C07146=1020.589,122.542,-113.459,167.523,51.122,159.470
C07147=1020.584,122.293,-113.440,167.519,51.128,159.471
C07148=1020.579,122.044,-113.421,167.517,51.134,159.471
C07149=1020.573,121.794,-113.402,167.514,51.141,159.472
C07150=1020.568,121.546,-113.383,167.511,51.148,159.473
C07151=1020.562,121.296,-113.363,167.508,51.155,159.474
C07152=1020.556,121.047,-113.344,167.505,51.160,159.475
C07153=1020.551,120.798,-113.325,167.502,51.167,159.475
C07154=1020.546,120.549,-113.306,167.500,51.174,159.476
C07155=1020.541,120.300,-113.287,167.497,51.180,159.477
C07156=1020.536,120.050,-113.267,167.494,51.187,159.478
C07157=1020.530,119.801,-113.248,167.491,51.193,159.478
C07158=1020.525,119.552,-113.229,167.488,51.200,159.479
C07159=1020.519,119.302,-113.210,167.485,51.207,159.480
C07160=1020.514,119.054,-113.191,167.482,51.214,159.481
C07161=1020.508,118.804,-113.172,167.479,51.219,159.482
C07162=1020.503,118.556,-113.153,167.476,51.226,159.482
C07163=1020.498,118.306,-113.134,167.474,51.233,159.483
C07164=1020.492,118.057,-113.114,167.470,51.240,159.484
C07165=1020.487,117.807,-113.096,167.468,51.246,159.485
C07166=1020.481,117.558,-113.077,167.464,51.253,159.485
C07167=1020.476,117.309,-113.058,167.462,51.259,159.486
C07168=1020.471,117.060,-113.039,167.459,51.266,159.487
C07169=1020.466,116.811,-113.019,167.456,51.272,159.488
C07170=1020.461,116.561,-113.000,167.453,51.278,159.489
C07171=1020.456,116.313,-112.981,167.450,51.285,159.489
C07172=1020.450,116.062,-112.963,167.447,51.291,159.490
C07173=1020.445,115.814,-112.944,167.444,51.298,159.491
C07174=1020.439,115.564,-112.925,167.442,51.305,159.492
C07175=1020.434,115.316,-112.906,167.439,51.311,159.492
C07176=1020.429,115.066,-112.887,167.436,51.317,159.493
C07177=1020.424,114.817,-112.868,167.433,51.324,159.494
C07178=1020.418,114.567,-112.849,167.430,51.331,159.495
C07179=1020.413,114.319,-112.830,167.427,51.337,159.495
C07180=1020.407,114.069,-112.811,167.424,51.344,159.496
C07181=1020.402,113.820,-112.792,167.422,51.350,159.497
C07182=1020.397,113.571,-112.773,167.419,51.356,159.498
C07183=1020.392,113.322,-112.755,167.416,51.363,159.498
C07184=1020.387,113.072,-112.735,167.413,51.370,159.499
C07185=1020.382,112.823,-112.716,167.411,51.376,159.500
C07186=1020.376,112.574,-112.697,167.407,51.383,159.501
C07187=1020.371,112.324,-112.679,167.405,51.389,159.502
C07188=1020.366,112.075,-112.659,167.401,51.395,159.502
C07189=1020.360,111.826,-112.642,167.399,51.402,159.503
C07190=1020.354,111.577,-112.623,167.395,51.409,159.504
C07191=1020.349,111.328,-112.604,167.393,51.415,159.505
C07192=1020.344,111.078,-112.585,167.390,51.422,159.505
C07193=1020.338,110.829,-112.567,167.387,51.428,159.506
C07194=1020.333,110.579,-112.548,167.385,51.435,159.507
C07195=1020.328,110.331,-112.530,167.382,51.442,159.508
C07196=1020.322,110.080,-112.511,167.379,51.448,159.509
C07197=1020.316,109.832,-112.493,167.376,51.455,159.509
C07198=1020.311,109.583,-112.474,167.373,51.461,159.510
C07199=1020.306,109.333,-112.455,167.370,51.468,159.511
C07200=1020.301,109.085,-112.436,167.368,51.475,159.512
C07201=1020.295,108.835,-112.418,167.364,51.482,159.512
C07202=1020.290,108.585,-112.400,167.362,51.488,159.513
C07203=1020.284,108.336,-112.382,167.359,51.495,159.514
C07204=1020.279,108.087,-112.364,167.356,51.502,159.515
C07205=1020.273,107.838,-112.344,167.353,51.508,159.516
C07206=1020.267,107.555,-112.324,167.350,51.516,159.517
C07207=1020.261,107.272,-112.303,167.347,51.523,159.518
C07208=1020.254,106.989,-112.282,167.344,51.531,159.518
C07209=1020.249,106.707,-112.262,167.341,51.539,159.519
C07210=1020.243,106.457,-112.243,167.337,51.545,159.520
C07211=1020.237,106.208,-112.225,167.335,51.551,159.521
C07212=1020.232,105.958,-112.206,167.332,51.558,159.522
C07213=1020.226,105.710,-112.188,167.329,51.565,159.523
C07214=1020.221,105.460,-112.170,167.326,51.572,159.523
C07215=1020.216,105.210,-112.151,167.324,51.579,159.524
C07216=1020.210,104.962,-112.133,167.321,51.584,159.525
C07217=1020.205,104.712,-112.115,167.318,51.591,159.526
C07218=1020.199,104.463,-112.097,167.316,51.598,159.526
C07219=1020.194,104.214,-112.078,167.312,51.605,159.527
C07220=1020.189,103.964,-112.060,167.310,51.611,159.528
C07221=1020.183,103.715,-112.042,167.306,51.618,159.529
C07222=1020.178,103.466,-112.023,167.304,51.624,159.530
C07223=1020.172,103.216,-112.005,167.302,51.631,159.530
C07224=1020.167,102.967,-111.987,167.298,51.638,159.531
C07225=1020.161,102.719,-111.969,167.296,51.644,159.532
C07226=1020.156,102.469,-111.950,167.292,51.651,159.533
C07227=1020.151,102.219,-111.932,167.290,51.658,159.533
C07228=1020.146,101.970,-111.915,167.288,51.664,159.534
C07229=1020.140,101.721,-111.895,167.284,51.670,159.535
C07230=1020.135,101.472,-111.878,167.282,51.677,159.536
C07231=1020.130,101.222,-111.860,167.279,51.684,159.537
C07232=1020.124,100.973,-111.842,167.276,51.691,159.537
C07233=1020.119,100.724,-111.823,167.274,51.697,159.538
C07234=1020.114,100.475,-111.805,167.270,51.704,159.539
C07235=1020.108,100.225,-111.787,167.268,51.710,159.540
C07236=1020.103,99.975,-111.768,167.266,51.717,159.541
C07237=1020.097,99.727,-111.750,167.262,51.723,159.541
C07238=1020.092,99.477,-111.732,167.260,51.730,159.542
C07239=1020.086,99.228,-111.714,167.257,51.737,159.543
C07240=1020.081,98.979,-111.696,167.254,51.743,159.544
C07241=1020.076,98.730,-111.678,167.252,51.749,159.544
C07242=1020.070,98.480,-111.660,167.248,51.756,159.545
C07243=1020.065,98.230,-111.642,167.246,51.763,159.546
C07244=1020.059,97.981,-111.625,167.243,51.770,159.547
C07245=1020.053,97.732,-111.607,167.241,51.776,159.548
C07246=1020.048,97.483,-111.589,167.237,51.783,159.548
C07247=1020.043,97.234,-111.570,167.235,51.790,159.549
C07248=1020.037,96.985,-111.553,167.231,51.796,159.550
C07249=1020.031,96.735,-111.535,167.229,51.803,159.551
C07250=1020.026,96.486,-111.517,167.227,51.810,159.552
C07251=1020.021,96.237,-111.499,167.224,51.817,159.552
C07252=1020.015,95.987,-111.481,167.221,51.823,159.553
C07253=1020.009,95.738,-111.464,167.218,51.830,159.554
C07254=1020.004,95.489,-111.445,167.215,51.836,159.555
C07255=1019.999,95.240,-111.428,167.213,51.843,159.556
C07256=1019.993,94.990,-111.410,167.210,51.850,159.556
C07257=1019.988,94.740,-111.392,167.208,51.857,159.557
C07258=1019.982,94.491,-111.374,167.204,51.863,159.558
C07259=1019.977,94.242,-111.357,167.202,51.869,159.559
C07260=1019.972,93.993,-111.340,167.200,51.876,159.559
C07261=1019.966,93.743,-111.321,167.196,51.883,159.560
C07262=1019.961,93.494,-111.304,167.194,51.890,159.561
C07263=1019.955,93.245,-111.286,167.190,51.896,159.562
C07264=1019.950,92.995,-111.268,167.188,51.903,159.563
C07265=1019.945,92.746,-111.250,167.186,51.909,159.563
C07266=1019.939,92.496,-111.232,167.183,51.916,159.564
C07267=1019.933,92.247,-111.215,167.180,51.922,159.565
C07268=1019.929,91.998,-111.197,167.177,51.929,159.566
C07269=1019.923,91.749,-111.179,167.175,51.936,159.567
C07270=1019.917,91.466,-111.159,167.171,51.943,159.567
C07271=1019.910,91.184,-111.139,167.169,51.951,159.568
C07272=1019.905,90.900,-111.119,167.166,51.958,159.569
C07273=1019.899,90.618,-111.099,167.162,51.965,159.570
C07274=1019.893,90.368,-111.081,167.159,51.972,159.571
C07275=1019.887,90.119,-111.064,167.157,51.979,159.572
C07276=1019.882,89.870,-111.045,167.154,51.985,159.572
C07277=1019.877,89.621,-111.028,167.151,51.992,159.573
C07278=1019.872,89.371,-111.011,167.149,51.999,159.574
C07279=1019.866,89.122,-110.993,167.146,52.005,159.575
C07280=1019.860,88.872,-110.975,167.143,52.012,159.575
C07281=1019.855,88.623,-110.958,167.141,52.018,159.576
C07282=1019.849,88.374,-110.941,167.139,52.025,159.577
C07283=1019.844,88.125,-110.923,167.135,52.032,159.578
C07284=1019.838,87.875,-110.906,167.133,52.039,159.579
C07285=1019.833,87.626,-110.889,167.130,52.046,159.580
C07286=1019.828,87.377,-110.871,167.127,52.052,159.580
C07287=1019.821,87.127,-110.854,167.124,52.059,159.581
C07288=1019.816,86.877,-110.837,167.122,52.065,159.582
C07289=1019.811,86.628,-110.819,167.120,52.072,159.583
C07290=1019.805,86.379,-110.802,167.116,52.079,159.583
C07291=1019.800,86.130,-110.785,167.114,52.085,159.584
C07292=1019.794,85.881,-110.767,167.111,52.092,159.585
C07293=1019.789,85.632,-110.750,167.108,52.099,159.586
C07294=1019.784,85.382,-110.733,167.106,52.106,159.587
C07295=1019.778,85.132,-110.715,167.103,52.113,159.587
C07296=1019.772,84.882,-110.698,167.100,52.119,159.588
C07297=1019.767,84.633,-110.680,167.097,52.126,159.589
C07298=1019.761,84.384,-110.663,167.095,52.132,159.590
C07299=1019.756,84.135,-110.646,167.093,52.139,159.591
C07300=1019.751,83.886,-110.628,167.089,52.145,159.591
C07301=1019.745,83.636,-110.612,167.087,52.152,159.592
C07302=1019.739,83.387,-110.595,167.085,52.159,159.593
C07303=1019.734,83.138,-110.578,167.081,52.166,159.594
C07304=1019.728,82.889,-110.560,167.079,52.172,159.594
C07305=1019.723,82.640,-110.543,167.076,52.179,159.595
C07306=1019.718,82.390,-110.526,167.073,52.185,159.596
C07307=1019.712,82.141,-110.508,167.071,52.192,159.597
C07308=1019.706,81.891,-110.491,167.068,52.198,159.597
C07309=1019.701,81.641,-110.473,167.065,52.205,159.598
C07310=1019.696,81.392,-110.457,167.063,52.212,159.599
C07311=1019.690,81.143,-110.439,167.060,52.218,159.600
C07312=1019.685,80.893,-110.422,167.057,52.225,159.601
C07313=1019.679,80.644,-110.405,167.055,52.232,159.602
C07314=1019.674,80.394,-110.388,167.052,52.239,159.602
C07315=1019.669,80.145,-110.370,167.049,52.245,159.603
C07316=1019.663,79.896,-110.353,167.047,52.251,159.604
C07317=1019.658,79.647,-110.336,167.044,52.258,159.605
C07318=1019.653,79.397,-110.319,167.041,52.264,159.605
C07319=1019.647,79.148,-110.301,167.039,52.271,159.606
C07320=1019.641,78.899,-110.285,167.036,52.278,159.607
C07321=1019.636,78.650,-110.267,167.033,52.284,159.608
C07322=1019.630,78.400,-110.251,167.031,52.291,159.608
C07323=1019.625,78.151,-110.233,167.028,52.297,159.609
C07324=1019.620,77.901,-110.216,167.026,52.304,159.610
C07325=1019.615,77.652,-110.199,167.023,52.311,159.611
C07326=1019.609,77.403,-110.182,167.021,52.317,159.611
C07327=1019.604,77.153,-110.165,167.018,52.324,159.612
C07328=1019.598,76.904,-110.147,167.015,52.330,159.613
C07329=1019.592,76.654,-110.131,167.013,52.336,159.614
C07330=1019.587,76.405,-110.114,167.010,52.343,159.615
C07331=1019.582,76.156,-110.097,167.007,52.350,159.615
C07332=1019.576,75.906,-110.080,167.004,52.357,159.616
C07333=1019.570,75.657,-110.064,167.002,52.363,159.617
C07334=1019.564,75.374,-110.045,166.999,52.371,159.618
C07335=1019.558,75.091,-110.026,166.996,52.379,159.619
C07336=1019.552,74.810,-110.006,166.993,52.386,159.620
C07337=1019.546,74.527,-109.987,166.990,52.394,159.621
C07338=1019.541,74.277,-109.970,166.987,52.401,159.621
C07339=1019.535,74.027,-109.954,166.984,52.407,159.622
C07340=1019.530,73.778,-109.937,166.982,52.413,159.623
C07341=1019.524,73.529,-109.920,166.979,52.421,159.624
C07342=1019.519,73.279,-109.903,166.977,52.427,159.624
C07343=1019.513,73.030,-109.887,166.974,52.433,159.625
C07344=1019.508,72.780,-109.870,166.971,52.440,159.626
C07345=1019.502,72.531,-109.853,166.969,52.447,159.627
C07346=1019.496,72.282,-109.836,166.965,52.453,159.627
C07347=1019.491,72.032,-109.819,166.963,52.460,159.628
C07348=1019.486,71.783,-109.802,166.961,52.467,159.629
C07349=1019.480,71.533,-109.786,166.958,52.473,159.630
C07350=1019.475,71.284,-109.770,166.955,52.480,159.631
C07351=1019.469,71.035,-109.753,166.953,52.487,159.631
C07352=1019.464,70.786,-109.736,166.950,52.493,159.632
C07353=1019.458,70.536,-109.719,166.948,52.500,159.633
C07354=1019.453,70.287,-109.703,166.945,52.507,159.634
C07355=1019.447,70.037,-109.686,166.942,52.513,159.634
C07356=1019.442,69.788,-109.669,166.940,52.520,159.635
C07357=1019.436,69.538,-109.653,166.938,52.526,159.636
C07358=1019.431,69.289,-109.636,166.934,52.533,159.637
C07359=1019.426,69.040,-109.620,166.932,52.540,159.637
C07360=1019.420,68.790,-109.603,166.930,52.546,159.638
C07361=1019.415,68.541,-109.586,166.926,52.553,159.639
C07362=1019.409,68.292,-109.569,166.924,52.559,159.640
C07363=1019.404,68.042,-109.552,166.922,52.566,159.641
C07364=1019.398,67.793,-109.536,166.918,52.573,159.641
C07365=1019.393,67.543,-109.519,166.916,52.579,159.642
C07366=1019.387,67.295,-109.503,166.914,52.586,159.643
C07367=1019.382,67.045,-109.487,166.910,52.592,159.644
C07368=1019.376,66.796,-109.470,166.908,52.599,159.644
C07369=1019.370,66.546,-109.455,166.906,52.606,159.645
C07370=1019.365,66.296,-109.438,166.903,52.612,159.646
C07371=1019.359,66.047,-109.422,166.900,52.619,159.647
C07372=1019.355,65.798,-109.405,166.898,52.626,159.648
C07373=1019.349,65.548,-109.389,166.895,52.632,159.648
C07374=1019.343,65.299,-109.372,166.893,52.639,159.649
C07375=1019.337,65.049,-109.356,166.891,52.646,159.650
C07376=1019.332,64.800,-109.339,166.887,52.653,159.651
C07377=1019.326,64.550,-109.323,166.885,52.659,159.651
C07378=1019.321,64.302,-109.307,166.882,52.666,159.652
C07379=1019.316,64.052,-109.290,166.880,52.673,159.653
C07380=1019.310,63.803,-109.274,166.877,52.679,159.654
C07381=1019.305,63.552,-109.258,166.874,52.686,159.654
C07382=1019.299,63.303,-109.241,166.871,52.692,159.655
C07383=1019.294,63.054,-109.225,166.869,52.699,159.656
C07384=1019.288,62.805,-109.209,166.866,52.706,159.657
C07385=1019.282,62.555,-109.192,166.864,52.713,159.658
C07386=1019.277,62.305,-109.177,166.860,52.719,159.658
C07387=1019.271,62.056,-109.161,166.858,52.726,159.659
C07388=1019.265,61.807,-109.145,166.856,52.733,159.660
C07389=1019.260,61.557,-109.129,166.853,52.740,159.661
C07390=1019.254,61.308,-109.113,166.851,52.746,159.662
C07391=1019.248,61.059,-109.097,166.848,52.754,159.662
C07392=1019.243,60.808,-109.080,166.845,52.760,159.663
C07393=1019.238,60.560,-109.065,166.842,52.767,159.664
C07394=1019.232,60.310,-109.048,166.840,52.774,159.665
C07395=1019.226,60.060,-109.033,166.838,52.780,159.666
C07396=1019.220,59.811,-109.016,166.835,52.787,159.666
C07397=1019.215,59.562,-109.001,166.832,52.793,159.667
C07398=1019.208,59.279,-108.983,166.830,52.801,159.668
C07399=1019.202,58.996,-108.964,166.826,52.810,159.669
C07400=1019.195,58.713,-108.946,166.823,52.817,159.670
C07401=1019.189,58.431,-108.928,166.820,52.825,159.671
C07402=1019.184,58.181,-108.912,166.818,52.831,159.672
C07403=1019.178,57.932,-108.896,166.815,52.838,159.672
C07404=1019.172,57.682,-108.880,166.812,52.845,159.673
C07405=1019.167,57.433,-108.864,166.809,52.852,159.674
C07406=1019.161,57.184,-108.848,166.807,52.858,159.675
C07407=1019.155,56.934,-108.833,166.805,52.865,159.675
C07408=1019.150,56.685,-108.817,166.802,52.872,159.676
C07409=1019.144,56.435,-108.801,166.800,52.878,159.677
C07410=1019.139,56.186,-108.785,166.796,52.885,159.677
C07411=1019.133,55.937,-108.770,166.794,52.892,159.678
C07412=1019.128,55.687,-108.754,166.792,52.898,159.679
C07413=1019.122,55.438,-108.737,166.788,52.905,159.680
C07414=1019.117,55.188,-108.722,166.786,52.912,159.681
C07415=1019.111,54.939,-108.705,166.784,52.918,159.682
C07416=1019.106,54.689,-108.690,166.781,52.925,159.682
C07417=1019.100,54.440,-108.674,166.779,52.932,159.683
C07418=1019.095,54.190,-108.658,166.775,52.939,159.684
C07419=1019.089,53.941,-108.642,166.773,52.945,159.684
C07420=1019.084,53.692,-108.627,166.771,52.952,159.685
C07421=1019.078,53.442,-108.611,166.768,52.959,159.686
C07422=1019.072,53.193,-108.595,166.765,52.965,159.687
C07423=1019.067,52.944,-108.579,166.763,52.972,159.688
C07424=1019.061,52.694,-108.564,166.760,52.979,159.688
C07425=1019.056,52.444,-108.547,166.758,52.985,159.689
C07426=1019.051,52.195,-108.532,166.755,52.992,159.690
C07427=1019.045,51.946,-108.515,166.752,52.998,159.690
C07428=1019.039,51.696,-108.500,166.750,53.005,159.691
C07429=1019.034,51.447,-108.484,166.747,53.012,159.692
C07430=1019.028,51.197,-108.468,166.744,53.018,159.693
C07431=1019.023,50.948,-108.453,166.742,53.025,159.694
C07432=1019.017,50.698,-108.437,166.739,53.032,159.694
C07433=1019.012,50.448,-108.421,166.737,53.038,159.695
C07434=1019.006,50.200,-108.406,166.735,53.045,159.696
C07435=1019.001,49.950,-108.390,166.731,53.052,159.697
C07436=1018.995,49.701,-108.374,166.729,53.058,159.697
C07437=1018.990,49.451,-108.359,166.727,53.064,159.698
C07438=1018.985,49.201,-108.342,166.724,53.072,159.699
C07439=1018.979,48.952,-108.327,166.721,53.078,159.700
C07440=1018.974,48.702,-108.311,166.719,53.085,159.700
C07441=1018.968,48.454,-108.295,166.715,53.091,159.701
C07442=1018.963,48.204,-108.280,166.713,53.098,159.702
C07443=1018.958,47.954,-108.264,166.711,53.104,159.703
C07444=1018.952,47.705,-108.248,166.708,53.111,159.703
C07445=1018.947,47.456,-108.233,166.705,53.117,159.704
C07446=1018.941,47.206,-108.217,166.703,53.124,159.705
C07447=1018.935,46.957,-108.201,166.701,53.130,159.706
C07448=1018.930,46.707,-108.186,166.698,53.137,159.706
C07449=1018.924,46.457,-108.170,166.695,53.143,159.707
C07450=1018.919,46.209,-108.155,166.693,53.150,159.708
C07451=1018.913,45.959,-108.139,166.690,53.157,159.708
C07452=1018.908,45.709,-108.124,166.688,53.164,159.709
C07453=1018.903,45.460,-108.107,166.685,53.170,159.710
C07454=1018.898,45.210,-108.092,166.682,53.177,159.711
C07455=1018.892,44.961,-108.076,166.680,53.183,159.711
C07456=1018.887,44.712,-108.060,166.678,53.190,159.712
C07457=1018.881,44.462,-108.045,166.675,53.196,159.713
C07458=1018.876,44.213,-108.030,166.672,53.202,159.713
C07459=1018.870,43.963,-108.013,166.670,53.209,159.714
C07460=1018.865,43.714,-107.998,166.667,53.215,159.715
C07461=1018.860,43.464,-107.983,166.664,53.222,159.716
C07462=1018.854,43.182,-107.965,166.661,53.230,159.717
C07463=1018.848,42.898,-107.947,166.658,53.237,159.717
C07464=1018.842,42.616,-107.930,166.655,53.244,159.718
C07465=1018.835,42.333,-107.912,166.653,53.252,159.719
C07466=1018.830,42.083,-107.897,166.650,53.258,159.720
C07467=1018.824,41.833,-107.881,166.648,53.265,159.721
C07468=1018.819,41.584,-107.866,166.644,53.271,159.721
C07469=1018.814,41.335,-107.852,166.642,53.278,159.722
C07470=1018.808,41.085,-107.836,166.640,53.284,159.723
C07471=1018.803,40.836,-107.820,166.637,53.292,159.723
C07472=1018.797,40.586,-107.805,166.635,53.298,159.724
C07473=1018.792,40.337,-107.790,166.632,53.305,159.725
C07474=1018.786,40.088,-107.775,166.629,53.312,159.726
C07475=1018.781,39.838,-107.759,166.627,53.318,159.726
C07476=1018.775,39.588,-107.744,166.624,53.325,159.727
C07477=1018.770,39.339,-107.729,166.621,53.331,159.728
C07478=1018.763,39.089,-107.714,166.619,53.338,159.729
C07479=1018.758,38.840,-107.699,166.616,53.345,159.729
C07480=1018.753,38.591,-107.683,166.614,53.351,159.730
C07481=1018.748,38.341,-107.668,166.611,53.358,159.731
C07482=1018.742,38.092,-107.653,166.608,53.365,159.732
C07483=1018.736,37.842,-107.638,166.606,53.371,159.732
C07484=1018.731,37.593,-107.623,166.604,53.378,159.733
C07485=1018.726,37.343,-107.607,166.600,53.384,159.734
C07486=1018.721,37.093,-107.592,166.598,53.391,159.735
C07487=1018.715,36.845,-107.577,166.596,53.397,159.735
C07488=1018.709,36.595,-107.562,166.593,53.404,159.736
C07489=1018.704,36.345,-107.547,166.591,53.411,159.737
C07490=1018.698,36.096,-107.532,166.587,53.418,159.738
C07491=1018.693,35.846,-107.517,166.585,53.424,159.738
C07492=1018.687,35.597,-107.503,166.583,53.431,159.739
C07493=1018.682,35.347,-107.487,166.580,53.437,159.740
C07494=1018.676,35.098,-107.472,166.578,53.444,159.741
C07495=1018.671,34.849,-107.457,166.575,53.451,159.741
C07496=1018.664,34.599,-107.442,166.572,53.458,159.742
C07497=1018.660,34.349,-107.428,166.569,53.465,159.743
C07498=1018.653,34.099,-107.413,166.567,53.471,159.743
C07499=1018.648,33.850,-107.398,166.565,53.478,159.744
C07500=1018.642,33.601,-107.383,166.561,53.484,159.745
C07501=1018.637,33.351,-107.368,166.559,53.491,159.746
C07502=1018.631,33.102,-107.354,166.556,53.498,159.746
C07503=1018.626,32.852,-107.339,166.554,53.504,159.747
C07504=1018.620,32.603,-107.324,166.552,53.511,159.748
C07505=1018.615,32.353,-107.309,166.548,53.518,159.749
C07506=1018.609,32.104,-107.295,166.546,53.525,159.749
C07507=1018.604,31.854,-107.279,166.543,53.531,159.750
C07508=1018.598,31.605,-107.265,166.541,53.538,159.751
C07509=1018.593,31.356,-107.249,166.538,53.544,159.752
C07510=1018.588,31.105,-107.235,166.535,53.552,159.752
C07511=1018.582,30.856,-107.220,166.533,53.558,159.753
C07512=1018.577,30.607,-107.205,166.530,53.565,159.754
C07513=1018.570,30.357,-107.190,166.528,53.571,159.754
C07514=1018.566,30.107,-107.175,166.525,53.577,159.755
C07515=1018.560,29.858,-107.161,166.522,53.584,159.756
C07516=1018.555,29.609,-107.146,166.520,53.591,159.757
C07517=1018.549,29.359,-107.131,166.518,53.598,159.757
C07518=1018.544,29.110,-107.116,166.514,53.604,159.758
C07519=1018.538,28.861,-107.102,166.512,53.611,159.759
C07520=1018.532,28.610,-107.087,166.509,53.617,159.759
C07521=1018.527,28.361,-107.072,166.507,53.624,159.760
C07522=1018.522,28.112,-107.057,166.505,53.630,159.761
C07523=1018.516,27.862,-107.043,166.501,53.637,159.761
C07524=1018.511,27.612,-107.028,166.499,53.644,159.762
C07525=1018.505,27.363,-107.013,166.497,53.650,159.763
C07526=1018.499,27.089,-106.997,166.494,53.658,159.764
C07527=1018.492,26.814,-106.981,166.491,53.665,159.765
C07528=1018.486,26.539,-106.965,166.488,53.673,159.766
C07529=1018.480,26.265,-106.949,166.485,53.680,159.766
C07530=1018.475,26.007,-106.935,166.482,53.687,159.767
C07531=1018.469,25.749,-106.919,166.479,53.694,159.768
C07532=1018.463,25.491,-106.904,166.477,53.701,159.769
C07533=1018.457,25.233,-106.890,166.474,53.708,159.769
C07534=1018.452,24.984,-106.875,166.471,53.714,159.770
C07535=1018.447,24.734,-106.861,166.468,53.721,159.771
C07536=1018.441,24.485,-106.846,166.466,53.727,159.771
C07537=1018.435,24.235,-106.832,166.463,53.735,159.772
C07538=1018.430,23.985,-106.817,166.461,53.741,159.773
C07539=1018.424,23.736,-106.803,166.459,53.748,159.774
C07540=1018.419,23.487,-106.788,166.455,53.754,159.774
C07541=1018.413,23.237,-106.774,166.453,53.761,159.775
C07542=1018.408,22.987,-106.760,166.450,53.768,159.776
C07543=1018.402,22.738,-106.745,166.448,53.775,159.777
C07544=1018.397,22.488,-106.731,166.444,53.781,159.777
C07545=1018.391,22.239,-106.717,166.443,53.788,159.778
C07546=1018.386,21.989,-106.702,166.440,53.794,159.779
C07547=1018.380,21.739,-106.688,166.437,53.802,159.779
C07548=1018.374,21.490,-106.673,166.435,53.808,159.780
C07549=1018.369,21.241,-106.659,166.431,53.814,159.781
C07550=1018.364,20.991,-106.644,166.429,53.821,159.782
C07551=1018.358,20.742,-106.630,166.427,53.827,159.782
C07552=1018.353,20.492,-106.616,166.424,53.835,159.783
C07553=1018.347,20.243,-106.602,166.422,53.841,159.784
C07554=1018.342,19.993,-106.587,166.419,53.848,159.784
C07555=1018.336,19.743,-106.573,166.416,53.854,159.785
C07556=1018.330,19.494,-106.559,166.414,53.860,159.786
C07557=1018.325,19.245,-106.545,166.411,53.868,159.786
C07558=1018.320,18.995,-106.530,166.409,53.874,159.787
C07559=1018.314,18.746,-106.516,166.406,53.881,159.788
C07560=1018.309,18.496,-106.502,166.403,53.887,159.789
C07561=1018.303,18.246,-106.488,166.400,53.894,159.789
C07562=1018.297,17.996,-106.474,166.398,53.901,159.790
C07563=1018.292,17.747,-106.459,166.394,53.908,159.791
C07564=1018.286,17.498,-106.445,166.393,53.914,159.791
C07565=1018.281,17.248,-106.431,166.390,53.921,159.792
C07566=1018.275,16.999,-106.418,166.387,53.928,159.793
C07567=1018.269,16.750,-106.403,166.385,53.934,159.794
C07568=1018.265,16.500,-106.389,166.382,53.941,159.794
C07569=1018.259,16.250,-106.375,166.380,53.948,159.795
C07570=1018.254,16.001,-106.361,166.376,53.954,159.795
C07571=1018.248,15.751,-106.347,166.374,53.961,159.796
C07572=1018.242,15.501,-106.333,166.371,53.968,159.797
C07573=1018.236,15.252,-106.318,166.369,53.975,159.798
C07574=1018.231,15.002,-106.304,166.367,53.981,159.798
C07575=1018.225,14.753,-106.290,166.363,53.987,159.799
C07576=1018.220,14.503,-106.277,166.361,53.994,159.800
C07577=1018.214,14.253,-106.263,166.358,54.001,159.800
C07578=1018.209,14.004,-106.249,166.355,54.007,159.801
C07579=1018.204,13.755,-106.234,166.352,54.014,159.802
C07580=1018.198,13.505,-106.220,166.350,54.021,159.803
C07581=1018.193,13.255,-106.206,166.348,54.027,159.803
C07582=1018.187,13.006,-106.192,166.345,54.034,159.804
C07583=1018.181,12.757,-106.179,166.343,54.041,159.805
C07584=1018.176,12.507,-106.165,166.339,54.048,159.805
C07585=1018.170,12.258,-106.151,166.337,54.055,159.806
C07586=1018.165,12.008,-106.137,166.334,54.061,159.807
C07587=1018.159,11.758,-106.123,166.331,54.069,159.808
C07588=1018.153,11.509,-106.110,166.329,54.075,159.808
C07589=1018.148,11.259,-106.097,166.326,54.082,159.809
C07590=1018.142,10.977,-106.081,166.323,54.089,159.810
C07591=1018.135,10.696,-106.066,166.320,54.097,159.811
C07592=1018.129,10.415,-106.050,166.318,54.105,159.812
C07593=1018.123,10.133,-106.035,166.314,54.112,159.812
C07594=1018.117,9.884,-106.021,166.311,54.119,159.813
C07595=1018.111,9.634,-106.007,166.308,54.126,159.814
C07596=1018.106,9.385,-105.994,166.306,54.132,159.814
C07597=1018.100,9.135,-105.980,166.303,54.140,159.815
C07598=1018.095,8.886,-105.966,166.301,54.146,159.816
C07599=1018.090,8.636,-105.953,166.298,54.153,159.816
C07600=1018.083,8.386,-105.939,166.296,54.159,159.817
C07601=1018.078,8.137,-105.926,166.293,54.167,159.818
C07602=1018.073,7.887,-105.912,166.290,54.173,159.819
C07603=1018.067,7.638,-105.898,166.287,54.179,159.819
C07604=1018.061,7.388,-105.885,166.285,54.186,159.820
C07605=1018.056,7.138,-105.871,166.282,54.193,159.820
C07606=1018.050,6.888,-105.858,166.280,54.200,159.821
C07607=1018.045,6.639,-105.844,166.276,54.207,159.822
C07608=1018.039,6.389,-105.830,166.274,54.213,159.823
C07609=1018.034,6.141,-105.817,166.271,54.220,159.823
C07610=1018.028,5.891,-105.803,166.269,54.226,159.824
C07611=1018.023,5.641,-105.790,166.265,54.233,159.825
C07612=1018.017,5.391,-105.776,166.264,54.240,159.825
C07613=1018.012,5.142,-105.762,166.260,54.247,159.826
C07614=1018.006,4.893,-105.749,166.258,54.253,159.827
C07615=1018.000,4.643,-105.735,166.255,54.260,159.827
C07616=1017.995,4.393,-105.722,166.253,54.266,159.828
C07617=1017.990,4.143,-105.708,166.250,54.273,159.829
C07618=1017.984,3.894,-105.694,166.247,54.280,159.829
C07619=1017.979,3.645,-105.681,166.245,54.286,159.830
C07620=1017.973,3.395,-105.668,166.242,54.293,159.831
C07621=1017.968,3.145,-105.654,166.240,54.300,159.832
C07622=1017.962,2.896,-105.640,166.236,54.306,159.832
C07623=1017.957,2.646,-105.628,166.234,54.313,159.833
C07624=1017.951,2.396,-105.614,166.231,54.320,159.834
C07625=1017.946,2.147,-105.600,166.229,54.326,159.834
C07626=1017.941,1.898,-105.587,166.225,54.333,159.835
C07627=1017.936,1.648,-105.573,166.223,54.339,159.835
C07628=1017.929,1.398,-105.560,166.220,54.346,159.836
C07629=1017.924,1.149,-105.546,166.218,54.353,159.837
C07630=1017.919,0.899,-105.533,166.215,54.359,159.837
C07631=1017.913,0.649,-105.519,166.212,54.366,159.838
C07632=1017.908,0.401,-105.506,166.210,54.373,159.839
C07633=1017.902,0.150,-105.493,166.207,54.379,159.839
C07634=1017.897,-0.099,-105.479,166.205,54.385,159.840
C07635=1017.891,-0.349,-105.466,166.201,54.392,159.841
C07636=1017.886,-0.599,-105.452,166.199,54.398,159.841
C07637=1017.881,-0.848,-105.439,166.196,54.406,159.842
C07638=1017.875,-1.097,-105.426,166.194,54.412,159.843
C07639=1017.870,-1.347,-105.412,166.192,54.418,159.843
C07640=1017.865,-1.597,-105.399,166.188,54.425,159.844
C07641=1017.859,-1.846,-105.386,166.186,54.431,159.845
C07642=1017.854,-2.096,-105.373,166.183,54.438,159.845
C07643=1017.848,-2.345,-105.359,166.181,54.445,159.846
C07644=1017.843,-2.595,-105.346,166.177,54.451,159.847
C07645=1017.838,-2.844,-105.333,166.175,54.458,159.847
C07646=1017.832,-3.094,-105.320,166.173,54.464,159.848
C07647=1017.827,-3.344,-105.306,166.169,54.471,159.848
C07648=1017.822,-3.594,-105.292,166.167,54.477,159.849
C07649=1017.817,-3.843,-105.279,166.164,54.484,159.850
C07650=1017.811,-4.092,-105.266,166.162,54.490,159.850
C07651=1017.805,-4.342,-105.253,166.158,54.497,159.851
C07652=1017.800,-4.593,-105.239,166.156,54.503,159.852
C07653=1017.794,-4.842,-105.226,166.153,54.510,159.852
C07654=1017.788,-5.121,-105.212,166.150,54.518,159.853
C07655=1017.782,-5.400,-105.197,166.148,54.525,159.854
C07656=1017.776,-5.680,-105.183,166.145,54.533,159.855
C07657=1017.770,-5.959,-105.169,166.141,54.541,159.855
C07658=1017.764,-6.209,-105.156,166.139,54.547,159.856
C07659=1017.758,-6.459,-105.143,166.136,54.554,159.857
C07660=1017.753,-6.709,-105.130,166.133,54.561,159.857
C07661=1017.748,-6.958,-105.117,166.130,54.567,159.858
C07662=1017.742,-7.208,-105.104,166.128,54.574,159.859
C07663=1017.736,-7.457,-105.091,166.125,54.581,159.859
C07664=1017.731,-7.706,-105.078,166.122,54.588,159.860
C07665=1017.725,-7.956,-105.065,166.119,54.594,159.861
C07666=1017.720,-8.206,-105.052,166.116,54.601,159.861
C07667=1017.715,-8.456,-105.040,166.114,54.607,159.862
C07668=1017.708,-8.705,-105.027,166.111,54.614,159.862
C07669=1017.703,-8.955,-105.014,166.109,54.621,159.863
C07670=1017.698,-9.204,-105.001,166.106,54.628,159.864
C07671=1017.693,-9.454,-104.988,166.103,54.634,159.865
C07672=1017.687,-9.704,-104.975,166.100,54.641,159.865
C07673=1017.681,-9.953,-104.963,166.098,54.648,159.866
C07674=1017.676,-10.203,-104.950,166.095,54.654,159.867
C07675=1017.671,-10.452,-104.937,166.093,54.661,159.867
C07676=1017.666,-10.702,-104.924,166.089,54.667,159.868
C07677=1017.659,-10.952,-104.911,166.086,54.675,159.868
C07678=1017.654,-11.201,-104.899,166.084,54.681,159.869
C07679=1017.649,-11.451,-104.886,166.081,54.688,159.870
C07680=1017.643,-11.701,-104.873,166.079,54.694,159.870
C07681=1017.638,-11.950,-104.860,166.075,54.701,159.871
C07682=1017.632,-12.200,-104.847,166.073,54.707,159.871
C07683=1017.627,-12.449,-104.835,166.070,54.714,159.872
C07684=1017.622,-12.699,-104.822,166.068,54.721,159.873
C07685=1017.616,-12.949,-104.809,166.064,54.727,159.873
C07686=1017.611,-13.198,-104.797,166.062,54.734,159.874
C07687=1017.605,-13.448,-104.784,166.059,54.740,159.875
C07688=1017.600,-13.698,-104.772,166.057,54.747,159.875
C07689=1017.595,-13.947,-104.758,166.054,54.754,159.876
C07690=1017.589,-14.196,-104.746,166.052,54.760,159.877
C07691=1017.583,-14.446,-104.733,166.048,54.767,159.877
C07692=1017.579,-14.696,-104.720,166.046,54.773,159.878
C07693=1017.573,-14.946,-104.708,166.043,54.780,159.878
C07694=1017.567,-15.195,-104.695,166.040,54.786,159.879
C07695=1017.562,-15.445,-104.682,166.037,54.793,159.880
C07696=1017.556,-15.695,-104.670,166.035,54.799,159.880
C07697=1017.552,-15.944,-104.657,166.031,54.806,159.881
C07698=1017.546,-16.194,-104.645,166.030,54.813,159.882
C07699=1017.541,-16.443,-104.632,166.026,54.820,159.882
C07700=1017.535,-16.693,-104.620,166.024,54.826,159.883
C07701=1017.529,-16.942,-104.608,166.021,54.833,159.883
C07702=1017.524,-17.192,-104.595,166.018,54.840,159.884
C07703=1017.518,-17.442,-104.583,166.016,54.846,159.885
C07704=1017.512,-17.691,-104.570,166.012,54.853,159.885
C07705=1017.508,-17.941,-104.558,166.010,54.859,159.886
C07706=1017.502,-18.191,-104.545,166.007,54.867,159.887
C07707=1017.497,-18.441,-104.534,166.004,54.874,159.887
C07708=1017.491,-18.690,-104.521,166.002,54.880,159.888
C07709=1017.486,-18.940,-104.509,165.998,54.887,159.888
C07710=1017.480,-19.190,-104.496,165.997,54.894,159.889
C07711=1017.474,-19.439,-104.484,165.993,54.900,159.890
C07712=1017.469,-19.689,-104.471,165.990,54.907,159.890
C07713=1017.463,-19.938,-104.459,165.988,54.913,159.891
C07714=1017.458,-20.188,-104.447,165.985,54.920,159.892
C07715=1017.453,-20.438,-104.435,165.983,54.927,159.892
C07716=1017.447,-20.688,-104.422,165.979,54.934,159.893
C07717=1017.442,-20.937,-104.410,165.977,54.940,159.894
C07718=1017.436,-21.214,-104.397,165.973,54.948,159.894
C07719=1017.430,-21.491,-104.383,165.971,54.955,159.895
C07720=1017.424,-21.770,-104.369,165.967,54.962,159.896
C07721=1017.418,-22.048,-104.356,165.965,54.970,159.896
C07722=1017.412,-22.297,-104.344,165.961,54.976,159.897
C07723=1017.406,-22.547,-104.331,165.959,54.983,159.897
C07724=1017.401,-22.796,-104.319,165.956,54.990,159.898
C07725=1017.396,-23.047,-104.307,165.954,54.996,159.899
C07726=1017.390,-23.296,-104.295,165.951,55.003,159.899
C07727=1017.386,-23.545,-104.282,165.947,55.010,159.900
C07728=1017.380,-23.795,-104.270,165.945,55.016,159.901
C07729=1017.375,-24.045,-104.258,165.942,55.023,159.901
C07730=1017.369,-24.294,-104.246,165.940,55.029,159.902
C07731=1017.364,-24.544,-104.233,165.936,55.036,159.902
C07732=1017.359,-24.794,-104.222,165.934,55.042,159.903
C07733=1017.353,-25.044,-104.209,165.931,55.049,159.903
C07734=1017.347,-25.293,-104.197,165.929,55.055,159.904
C07735=1017.342,-25.542,-104.185,165.925,55.062,159.905
C07736=1017.336,-25.792,-104.173,165.923,55.068,159.905
C07737=1017.331,-26.042,-104.161,165.920,55.075,159.906
C07738=1017.326,-26.291,-104.149,165.918,55.081,159.906
C07739=1017.321,-26.542,-104.136,165.914,55.088,159.907
C07740=1017.316,-26.791,-104.124,165.911,55.095,159.907
C07741=1017.310,-27.040,-104.112,165.909,55.101,159.908
C07742=1017.305,-27.291,-104.100,165.905,55.108,159.909
C07743=1017.299,-27.540,-104.088,165.903,55.114,159.909
C07744=1017.294,-27.790,-104.076,165.900,55.122,159.910
C07745=1017.288,-28.039,-104.064,165.898,55.128,159.911
C07746=1017.283,-28.289,-104.052,165.895,55.135,159.911
C07747=1017.277,-28.538,-104.041,165.892,55.141,159.912
C07748=1017.272,-28.789,-104.029,165.889,55.148,159.912
C07749=1017.267,-29.038,-104.017,165.886,55.155,159.913
C07750=1017.262,-29.288,-104.005,165.884,55.162,159.914
C07751=1017.257,-29.537,-103.994,165.881,55.168,159.914
C07752=1017.250,-29.787,-103.982,165.878,55.175,159.915
C07753=1017.245,-30.037,-103.970,165.876,55.181,159.916
C07754=1017.240,-30.286,-103.958,165.872,55.188,159.916
C07755=1017.234,-30.536,-103.946,165.869,55.195,159.917
C07756=1017.229,-30.786,-103.934,165.867,55.201,159.917
C07757=1017.223,-31.035,-103.923,165.864,55.208,159.918
C07758=1017.218,-31.285,-103.912,165.862,55.215,159.919
C07759=1017.212,-31.535,-103.899,165.859,55.222,159.919
C07760=1017.207,-31.785,-103.888,165.855,55.229,159.920
C07761=1017.202,-32.034,-103.876,165.853,55.235,159.920
C07762=1017.196,-32.283,-103.865,165.850,55.242,159.921
C07763=1017.191,-32.533,-103.853,165.847,55.248,159.921
C07764=1017.185,-32.783,-103.841,165.845,55.255,159.922
C07765=1017.180,-33.033,-103.829,165.841,55.261,159.923
C07766=1017.175,-33.283,-103.818,165.839,55.268,159.923
C07767=1017.169,-33.531,-103.806,165.836,55.275,159.924
C07768=1017.164,-33.781,-103.795,165.833,55.281,159.924
C07769=1017.158,-34.032,-103.783,165.830,55.288,159.925
C07770=1017.153,-34.281,-103.771,165.827,55.294,159.925
C07771=1017.147,-34.530,-103.760,165.825,55.301,159.926
C07772=1017.142,-34.780,-103.748,165.822,55.308,159.927
C07773=1017.137,-35.029,-103.736,165.819,55.314,159.927
C07774=1017.131,-35.280,-103.724,165.816,55.321,159.928
C07775=1017.126,-35.530,-103.713,165.813,55.327,159.928
C07776=1017.121,-35.779,-103.702,165.811,55.334,159.929
C07777=1017.115,-36.028,-103.690,165.807,55.341,159.929
C07778=1017.110,-36.278,-103.678,165.805,55.347,159.930
C07779=1017.105,-36.528,-103.667,165.802,55.354,159.931
C07780=1017.100,-36.778,-103.655,165.800,55.360,159.931
C07781=1017.094,-37.027,-103.643,165.797,55.367,159.932
C07782=1017.088,-37.304,-103.631,165.794,55.374,159.933
C07783=1017.083,-37.581,-103.618,165.791,55.381,159.933
C07784=1017.076,-37.857,-103.605,165.787,55.389,159.934
C07785=1017.071,-38.134,-103.592,165.784,55.396,159.934
C07786=1017.066,-38.384,-103.581,165.781,55.402,159.935
C07787=1017.060,-38.633,-103.569,165.778,55.409,159.935
C07788=1017.055,-38.882,-103.558,165.776,55.415,159.936
C07789=1017.050,-39.132,-103.546,165.773,55.422,159.936
C07790=1017.044,-39.383,-103.535,165.771,55.428,159.937
C07791=1017.039,-39.632,-103.524,165.767,55.435,159.938
C07792=1017.034,-39.882,-103.512,165.764,55.442,159.938
C07793=1017.028,-40.132,-103.501,165.762,55.448,159.939
C07794=1017.023,-40.381,-103.490,165.759,55.455,159.939
C07795=1017.017,-40.631,-103.479,165.755,55.462,159.940
C07796=1017.012,-40.881,-103.468,165.753,55.468,159.940
C07797=1017.006,-41.130,-103.457,165.750,55.475,159.941
C07798=1017.001,-41.380,-103.445,165.747,55.482,159.941
C07799=1016.996,-41.629,-103.434,165.745,55.488,159.942
C07800=1016.991,-41.879,-103.423,165.741,55.495,159.943
C07801=1016.985,-42.129,-103.412,165.738,55.502,159.943
C07802=1016.980,-42.379,-103.401,165.736,55.508,159.944
C07803=1016.974,-42.628,-103.390,165.733,55.515,159.944
C07804=1016.969,-42.878,-103.378,165.729,55.522,159.945
C07805=1016.963,-43.127,-103.367,165.727,55.528,159.945
C07806=1016.958,-43.377,-103.356,165.724,55.535,159.946
C07807=1016.953,-43.627,-103.345,165.722,55.541,159.947
C07808=1016.948,-43.876,-103.333,165.719,55.548,159.947
C07809=1016.942,-44.126,-103.323,165.715,55.555,159.948
C07810=1016.937,-44.376,-103.311,165.713,55.561,159.948
C07811=1016.932,-44.626,-103.301,165.710,55.568,159.949
C07812=1016.927,-44.876,-103.290,165.707,55.575,159.949
C07813=1016.921,-45.125,-103.279,165.705,55.581,159.950
C07814=1016.916,-45.375,-103.267,165.701,55.588,159.950
C07815=1016.910,-45.624,-103.256,165.699,55.594,159.951
C07816=1016.905,-45.874,-103.245,165.696,55.601,159.952
C07817=1016.899,-46.124,-103.234,165.693,55.608,159.952
C07818=1016.894,-46.373,-103.222,165.691,55.614,159.953
C07819=1016.889,-46.624,-103.212,165.687,55.621,159.953
C07820=1016.884,-46.873,-103.201,165.685,55.627,159.954
C07821=1016.878,-47.123,-103.190,165.682,55.634,159.954
C07822=1016.873,-47.373,-103.178,165.678,55.640,159.955
C07823=1016.867,-47.622,-103.168,165.676,55.647,159.955
C07824=1016.863,-47.873,-103.157,165.673,55.654,159.956
C07825=1016.857,-48.122,-103.146,165.671,55.660,159.957
C07826=1016.853,-48.371,-103.135,165.668,55.667,159.957
C07827=1016.847,-48.621,-103.124,165.665,55.673,159.958
C07828=1016.842,-48.870,-103.113,165.662,55.679,159.958
C07829=1016.836,-49.121,-103.102,165.659,55.686,159.958
C07830=1016.831,-49.370,-103.091,165.656,55.692,159.959
C07831=1016.826,-49.620,-103.080,165.653,55.699,159.960
C07832=1016.820,-49.869,-103.069,165.651,55.706,159.960
C07833=1016.815,-50.120,-103.058,165.647,55.712,159.961
///RCONF 1,0,0,1,0,0,0,0,0,0,0,0,0,0,0,0,0,0,0,0,0,0,0,0
C07834=1016.810,-50.369,-103.047,165.645,55.718,159.961
C07835=1016.805,-50.619,-103.036,165.642,55.725,159.962
C07836=1016.800,-50.870,-103.025,165.639,55.732,159.962
C07837=1016.795,-51.118,-103.015,165.637,55.738,159.963
C07838=1016.789,-51.368,-103.004,165.633,55.745,159.963
C07839=1016.784,-51.618,-102.994,165.630,55.752,159.964
C07840=1016.778,-51.867,-102.983,165.628,55.758,159.965
C07841=1016.772,-52.118,-102.973,165.625,55.765,159.965
C07842=1016.767,-52.367,-102.962,165.622,55.772,159.966
C07843=1016.761,-52.617,-102.952,165.618,55.779,159.966
C07844=1016.757,-52.866,-102.941,165.616,55.785,159.967
C07845=1016.751,-53.116,-102.930,165.613,55.792,159.967
C07846=1016.745,-53.394,-102.919,165.610,55.799,159.968
C07847=1016.739,-53.670,-102.907,165.606,55.807,159.968
C07848=1016.733,-53.947,-102.896,165.603,55.814,159.969
C07849=1016.727,-54.224,-102.885,165.601,55.822,159.970
C07850=1016.721,-54.474,-102.874,165.598,55.829,159.970
C07851=1016.716,-54.724,-102.863,165.594,55.835,159.971
C07852=1016.711,-54.973,-102.852,165.591,55.842,159.971
C07853=1016.706,-55.223,-102.842,165.589,55.849,159.972
C07854=1016.700,-55.473,-102.832,165.586,55.855,159.972
C07855=1016.695,-55.723,-102.821,165.583,55.862,159.973
C07856=1016.689,-55.973,-102.811,165.581,55.869,159.974
C07857=1016.684,-56.222,-102.801,165.577,55.876,159.974
C07858=1016.679,-56.472,-102.790,165.574,55.882,159.975
C07859=1016.673,-56.722,-102.780,165.571,55.889,159.975
C07860=1016.668,-56.971,-102.769,165.568,55.895,159.975
C07861=1016.663,-57.221,-102.760,165.565,55.902,159.976
C07862=1016.657,-57.471,-102.749,165.562,55.909,159.976
C07863=1016.652,-57.720,-102.739,165.560,55.915,159.977
C07864=1016.647,-57.970,-102.729,165.557,55.922,159.978
C07865=1016.641,-58.220,-102.719,165.554,55.929,159.978
C07866=1016.636,-58.470,-102.707,165.551,55.935,159.979
C07867=1016.631,-58.720,-102.697,165.548,55.942,159.979
C07868=1016.626,-58.969,-102.687,165.545,55.949,159.980
C07869=1016.621,-59.219,-102.677,165.543,55.955,159.980
C07870=1016.615,-59.469,-102.666,165.539,55.961,159.981
C07871=1016.610,-59.718,-102.656,165.536,55.968,159.981
C07872=1016.605,-59.968,-102.646,165.534,55.975,159.982
C07873=1016.599,-60.218,-102.635,165.531,55.981,159.982
C07874=1016.594,-60.467,-102.626,165.528,55.988,159.983
C07875=1016.589,-60.717,-102.615,165.525,55.995,159.984
C07876=1016.583,-60.967,-102.605,165.522,56.001,159.984
C07877=1016.578,-61.216,-102.595,165.520,56.007,159.984
C07878=1016.573,-61.466,-102.585,165.517,56.014,159.985
C07879=1016.568,-61.716,-102.575,165.513,56.021,159.985
C07880=1016.562,-61.966,-102.565,165.511,56.027,159.986
C07881=1016.557,-62.216,-102.554,165.508,56.033,159.986
C07882=1016.552,-62.465,-102.544,165.504,56.040,159.987
C07883=1016.546,-62.715,-102.534,165.502,56.047,159.987
C07884=1016.541,-62.965,-102.524,165.499,56.054,159.988
C07885=1016.537,-63.215,-102.513,165.496,56.059,159.988
C07886=1016.531,-63.465,-102.503,165.493,56.066,159.989
C07887=1016.527,-63.714,-102.493,165.490,56.073,159.989
C07888=1016.521,-63.964,-102.482,165.488,56.079,159.990
C07889=1016.515,-64.214,-102.472,165.484,56.086,159.990
C07890=1016.511,-64.463,-102.462,165.481,56.092,159.991
C07891=1016.505,-64.713,-102.452,165.479,56.099,159.991
C07892=1016.500,-64.963,-102.442,165.476,56.106,159.992
C07893=1016.495,-65.213,-102.432,165.473,56.111,159.992
C07894=1016.490,-65.462,-102.422,165.470,56.118,159.993
C07895=1016.484,-65.712,-102.412,165.468,56.125,159.993
C07896=1016.479,-65.961,-102.402,165.464,56.131,159.994
C07897=1016.474,-66.211,-102.392,165.461,56.138,159.994
C07898=1016.469,-66.461,-102.382,165.459,56.144,159.995
C07899=1016.464,-66.711,-102.372,165.455,56.150,159.995
C07900=1016.458,-66.961,-102.362,165.453,56.157,159.996
C07901=1016.453,-67.210,-102.352,165.450,56.164,159.996
C07902=1016.448,-67.460,-102.342,165.448,56.169,159.997
C07903=1016.443,-67.710,-102.332,165.444,56.176,159.997
C07904=1016.438,-67.960,-102.322,165.441,56.182,159.997
C07905=1016.433,-68.209,-102.312,165.439,56.189,159.998
C07906=1016.428,-68.459,-102.302,165.435,56.196,159.998
C07907=1016.423,-68.709,-102.292,165.433,56.201,159.999
C07908=1016.418,-68.958,-102.282,165.430,56.208,159.999
C07909=1016.412,-69.208,-102.272,165.427,56.214,160.000
C07910=1016.408,-69.486,-102.261,165.424,56.222,160.001
C07911=1016.401,-69.764,-102.249,165.420,56.229,160.001
C07912=1016.396,-70.042,-102.238,165.417,56.236,160.001
C07913=1016.389,-70.321,-102.227,165.414,56.243,160.002
C07914=1016.385,-70.570,-102.217,165.412,56.249,160.002
C07915=1016.380,-70.820,-102.208,165.408,56.255,160.003
C07916=1016.374,-71.070,-102.197,165.405,56.262,160.003
C07917=1016.370,-71.319,-102.188,165.402,56.268,160.004
C07918=1016.364,-71.569,-102.177,165.399,56.275,160.004
C07919=1016.359,-71.819,-102.168,165.397,56.280,160.004
C07920=1016.354,-72.069,-102.158,165.394,56.287,160.005
C07921=1016.349,-72.319,-102.148,165.391,56.293,160.005
C07922=1016.345,-72.568,-102.139,165.388,56.300,160.006
C07923=1016.339,-72.818,-102.128,165.385,56.306,160.006
C07924=1016.335,-73.068,-102.118,165.382,56.313,160.007
C07925=1016.330,-73.317,-102.108,165.379,56.318,160.007
C07926=1016.325,-73.568,-102.098,165.377,56.324,160.008
C07927=1016.320,-73.817,-102.088,165.374,56.331,160.008
C07928=1016.314,-74.067,-102.078,165.371,56.337,160.008
C07929=1016.310,-74.317,-102.069,165.368,56.344,160.009
C07930=1016.305,-74.567,-102.059,165.365,56.349,160.009
C07931=1016.299,-74.816,-102.050,165.362,56.356,160.010
C07932=1016.294,-75.066,-102.040,165.358,56.362,160.010
C07933=1016.290,-75.316,-102.031,165.356,56.369,160.011
C07934=1016.283,-75.566,-102.021,165.353,56.376,160.011
C07935=1016.279,-75.815,-102.011,165.351,56.381,160.012
C07936=1016.274,-76.065,-102.002,165.348,56.388,160.012
C07937=1016.269,-76.315,-101.992,165.344,56.395,160.013
C07938=1016.263,-76.564,-101.983,165.342,56.401,160.013
C07939=1016.259,-76.814,-101.974,165.339,56.408,160.013
C07940=1016.253,-77.064,-101.964,165.336,56.414,160.014
C07941=1016.248,-77.314,-101.955,165.333,56.420,160.014
C07942=1016.243,-77.563,-101.945,165.330,56.427,160.015
C07943=1016.238,-77.814,-101.935,165.327,56.433,160.015
C07944=1016.233,-78.064,-101.926,165.324,56.440,160.016
C07945=1016.227,-78.313,-101.917,165.322,56.446,160.016
C07946=1016.223,-78.563,-101.908,165.318,56.453,160.017
C07947=1016.217,-78.813,-101.898,165.316,56.458,160.017
C07948=1016.212,-79.062,-101.889,165.313,56.465,160.017
C07949=1016.207,-79.312,-101.879,165.309,56.471,160.018
C07950=1016.203,-79.561,-101.870,165.307,56.478,160.018
C07951=1016.197,-79.812,-101.861,165.303,56.484,160.019
C07952=1016.192,-80.061,-101.851,165.301,56.491,160.019
C07953=1016.187,-80.311,-101.842,165.298,56.497,160.019
C07954=1016.182,-80.560,-101.833,165.296,56.503,160.020
C07955=1016.177,-80.811,-101.823,165.292,56.510,160.021
C07956=1016.171,-81.061,-101.815,165.289,56.517,160.021
C07957=1016.167,-81.310,-101.805,165.287,56.523,160.021
C07958=1016.161,-81.560,-101.797,165.284,56.530,160.022
C07959=1016.156,-81.809,-101.787,165.281,56.537,160.022
C07960=1016.151,-82.060,-101.778,165.278,56.542,160.023
C07961=1016.145,-82.309,-101.769,165.275,56.549,160.023
C07962=1016.140,-82.559,-101.760,165.272,56.556,160.024
C07963=1016.135,-82.809,-101.751,165.269,56.562,160.024
C07964=1016.131,-83.059,-101.742,165.266,56.569,160.025
C07965=1016.125,-83.309,-101.733,165.263,56.576,160.025
C07966=1016.120,-83.558,-101.723,165.260,56.582,160.026
C07967=1016.115,-83.808,-101.715,165.257,56.589,160.026
C07968=1016.109,-84.058,-101.706,165.255,56.594,160.026
C07969=1016.105,-84.307,-101.697,165.252,56.601,160.027
C07970=1016.099,-84.557,-101.688,165.248,56.608,160.027
C07971=1016.095,-84.807,-101.679,165.246,56.614,160.028
C07972=1016.089,-85.057,-101.670,165.243,56.621,160.028
C07973=1016.084,-85.307,-101.660,165.240,56.627,160.029
C07974=1016.079,-85.587,-101.651,165.237,56.635,160.029
C07975=1016.073,-85.867,-101.641,165.233,56.642,160.030
C07976=1016.067,-86.147,-101.631,165.230,56.648,160.030
C07977=1016.061,-86.426,-101.621,165.226,56.656,160.030
C07978=1016.057,-86.676,-101.612,165.224,56.662,160.031
C07979=1016.051,-86.927,-101.603,165.221,56.669,160.031
C07980=1016.046,-87.176,-101.594,165.219,56.675,160.032
C07981=1016.041,-87.426,-101.585,165.215,56.681,160.032
C07982=1016.035,-87.675,-101.576,165.213,56.688,160.033
C07983=1016.031,-87.925,-101.567,165.209,56.694,160.033
C07984=1016.026,-88.175,-101.559,165.206,56.701,160.034
C07985=1016.020,-88.425,-101.550,165.204,56.707,160.034
C07986=1016.016,-88.675,-101.541,165.200,56.714,160.034
C07987=1016.011,-88.925,-101.533,165.198,56.719,160.035
C07988=1016.006,-89.175,-101.523,165.195,56.726,160.035
C07989=1016.000,-89.424,-101.514,165.192,56.732,160.036
C07990=1015.996,-89.674,-101.505,165.189,56.738,160.036
C07991=1015.991,-89.924,-101.497,165.187,56.745,160.037
C07992=1015.985,-90.173,-101.488,165.183,56.751,160.037
C07993=1015.981,-90.423,-101.479,165.181,56.757,160.038
C07994=1015.976,-90.673,-101.471,165.177,56.764,160.038
C07995=1015.971,-90.923,-101.462,165.175,56.770,160.038
C07996=1015.966,-91.173,-101.453,165.172,56.776,160.039
C07997=1015.961,-91.422,-101.445,165.169,56.782,160.039
C07998=1015.956,-91.672,-101.436,165.166,56.789,160.039
C07999=1015.951,-91.922,-101.427,165.163,56.795,160.040
C08000=1015.946,-92.172,-101.417,165.160,56.801,160.040
C08001=1015.941,-92.421,-101.409,165.158,56.808,160.041
C08002=1015.935,-92.671,-101.400,165.154,56.814,160.041
C08003=1015.931,-92.921,-101.391,165.152,56.820,160.041
C08004=1015.926,-93.171,-101.383,165.148,56.827,160.042
C08005=1015.920,-93.420,-101.374,165.146,56.832,160.042
C08006=1015.916,-93.671,-101.365,165.142,56.839,160.042
C08007=1015.911,-93.920,-101.357,165.140,56.845,160.043
C08008=1015.906,-94.170,-101.348,165.137,56.851,160.043
C08009=1015.901,-94.420,-101.339,165.134,56.857,160.044
C08010=1015.896,-94.670,-101.331,165.131,56.864,160.044
C08011=1015.891,-94.920,-101.322,165.128,56.870,160.045
C08012=1015.886,-95.169,-101.313,165.125,56.876,160.045
C08013=1015.882,-95.419,-101.305,165.122,56.882,160.045
C08014=1015.877,-95.669,-101.297,165.120,56.888,160.046
C08015=1015.872,-95.919,-101.288,165.117,56.895,160.046
C08016=1015.867,-96.169,-101.279,165.114,56.900,160.046
C08017=1015.862,-96.419,-101.270,165.110,56.907,160.047
C08018=1015.857,-96.669,-101.261,165.108,56.913,160.047
C08019=1015.852,-96.918,-101.253,165.105,56.919,160.047
C08020=1015.847,-97.167,-101.245,165.102,56.925,160.048
C08021=1015.843,-97.417,-101.236,165.100,56.931,160.048
C08022=1015.838,-97.667,-101.227,165.096,56.937,160.048
C08023=1015.833,-97.917,-101.218,165.094,56.944,160.049
C08024=1015.828,-98.167,-101.210,165.090,56.950,160.049
C08025=1015.823,-98.417,-101.202,165.088,56.956,160.050
C08026=1015.818,-98.667,-101.193,165.085,56.963,160.050
C08027=1015.813,-98.916,-101.186,165.082,56.969,160.051
C08028=1015.808,-99.166,-101.178,165.079,56.975,160.051
C08029=1015.803,-99.416,-101.169,165.077,56.981,160.051
C08030=1015.797,-99.666,-101.161,165.073,56.987,160.052
C08031=1015.792,-99.916,-101.153,165.071,56.994,160.052
C08032=1015.788,-100.166,-101.144,165.067,57.000,160.052
C08033=1015.783,-100.415,-101.136,165.065,57.006,160.053
C08034=1015.778,-100.665,-101.128,165.062,57.013,160.053
C08035=1015.773,-100.915,-101.119,165.059,57.019,160.054
C08036=1015.768,-101.165,-101.112,165.056,57.025,160.054
C08037=1015.763,-101.414,-101.103,165.054,57.032,160.055
C08038=1015.758,-101.697,-101.094,165.051,57.039,160.055
C08039=1015.752,-101.978,-101.085,165.047,57.046,160.055
C08040=1015.746,-102.261,-101.076,165.043,57.052,160.056
C08041=1015.741,-102.543,-101.067,165.040,57.059,160.056
C08042=1015.736,-102.793,-101.058,165.038,57.066,160.057
C08043=1015.731,-103.042,-101.050,165.034,57.072,160.057
C08044=1015.726,-103.293,-101.042,165.032,57.078,160.057
C08045=1015.721,-103.542,-101.034,165.028,57.084,160.057
C08046=1015.716,-103.792,-101.026,165.026,57.091,160.058
C08047=1015.711,-104.042,-101.017,165.023,57.097,160.058
C08048=1015.706,-104.292,-101.010,165.020,57.103,160.059
C08049=1015.702,-104.541,-101.001,165.017,57.108,160.059
C08050=1015.697,-104.792,-100.993,165.014,57.115,160.060
C08051=1015.692,-105.042,-100.985,165.012,57.121,160.060
C08052=1015.687,-105.291,-100.977,165.008,57.127,160.060
C08053=1015.682,-105.541,-100.969,165.006,57.133,160.061
C08054=1015.677,-105.791,-100.961,165.002,57.140,160.061
C08055=1015.673,-106.040,-100.953,165.000,57.146,160.061
C08056=1015.668,-106.291,-100.945,164.998,57.152,160.062
C08057=1015.662,-106.540,-100.937,164.994,57.158,160.062
C08058=1015.658,-106.790,-100.929,164.992,57.164,160.062
C08059=1015.653,-107.040,-100.921,164.988,57.170,160.063
C08060=1015.648,-107.290,-100.913,164.985,57.176,160.063
C08061=1015.643,-107.539,-100.905,164.983,57.183,160.064
C08062=1015.638,-107.789,-100.897,164.980,57.189,160.064
C08063=1015.633,-108.040,-100.889,164.977,57.195,160.064
C08064=1015.629,-108.289,-100.881,164.974,57.201,160.064
C08065=1015.624,-108.539,-100.873,164.972,57.208,160.065
C08066=1015.619,-108.789,-100.866,164.968,57.214,160.065
C08067=1015.614,-109.038,-100.858,164.966,57.220,160.066
C08068=1015.609,-109.289,-100.850,164.963,57.225,160.066
C08069=1015.604,-109.538,-100.843,164.959,57.232,160.066
C08070=1015.599,-109.788,-100.835,164.958,57.238,160.067
C08071=1015.594,-110.037,-100.827,164.954,57.245,160.067
C08072=1015.589,-110.288,-100.819,164.951,57.250,160.067
C08073=1015.585,-110.537,-100.812,164.948,57.257,160.068
C08074=1015.580,-110.787,-100.803,164.945,57.262,160.068
C08075=1015.575,-111.037,-100.796,164.943,57.268,160.068
C08076=1015.570,-111.287,-100.788,164.940,57.275,160.069
C08077=1015.565,-111.537,-100.781,164.937,57.281,160.069
C08078=1015.560,-111.786,-100.773,164.934,57.287,160.069
C08079=1015.555,-112.036,-100.765,164.931,57.293,160.070
C08080=1015.551,-112.286,-100.758,164.929,57.299,160.070
C08081=1015.546,-112.536,-100.750,164.925,57.305,160.070
C08082=1015.541,-112.785,-100.742,164.922,57.311,160.071
C08083=1015.536,-113.036,-100.734,164.921,57.318,160.071
C08084=1015.532,-113.285,-100.727,164.917,57.324,160.072
C08085=1015.526,-113.535,-100.720,164.914,57.330,160.072
C08086=1015.522,-113.785,-100.712,164.912,57.336,160.072
C08087=1015.516,-114.035,-100.704,164.908,57.342,160.073
C08088=1015.512,-114.284,-100.696,164.906,57.348,160.073
C08089=1015.507,-114.535,-100.689,164.903,57.354,160.073
C08090=1015.503,-114.784,-100.681,164.900,57.360,160.074
C08091=1015.497,-115.034,-100.674,164.897,57.366,160.074
C08092=1015.493,-115.284,-100.667,164.894,57.372,160.074
C08093=1015.488,-115.534,-100.659,164.891,57.378,160.075
C08094=1015.483,-115.784,-100.651,164.889,57.384,160.075
C08095=1015.479,-116.034,-100.644,164.886,57.391,160.075
C08096=1015.473,-116.284,-100.637,164.883,57.397,160.076
C08097=1015.469,-116.533,-100.629,164.881,57.402,160.076
C08098=1015.464,-116.784,-100.622,164.877,57.409,160.076
C08099=1015.460,-117.033,-100.614,164.874,57.414,160.077
C08100=1015.454,-117.283,-100.607,164.872,57.420,160.077
C08101=1015.450,-117.533,-100.600,164.868,57.427,160.077
C08102=1015.445,-117.768,-100.592,164.866,57.432,160.078
C08103=1015.441,-118.003,-100.586,164.863,57.438,160.078
C08104=1015.436,-118.237,-100.579,164.860,57.443,160.078
C08105=1015.432,-118.473,-100.572,164.858,57.449,160.079
C08106=1015.427,-118.707,-100.565,164.855,57.455,160.079
C08107=1015.422,-118.942,-100.558,164.852,57.460,160.079
C08108=1015.418,-119.177,-100.551,164.850,57.466,160.079
C08109=1015.413,-119.412,-100.544,164.847,57.472,160.080
C08110=1015.408,-119.662,-100.537,164.845,57.478,160.080
C08111=1015.404,-119.911,-100.529,164.842,57.484,160.081
C08112=1015.399,-120.162,-100.522,164.839,57.490,160.081
C08113=1015.394,-120.412,-100.515,164.836,57.496,160.081
C08114=1015.390,-120.661,-100.508,164.834,57.502,160.082
C08115=1015.385,-120.911,-100.500,164.831,57.507,160.082
C08116=1015.380,-121.161,-100.493,164.828,57.514,160.082
C08117=1015.375,-121.410,-100.486,164.825,57.520,160.082
C08118=1015.370,-121.723,-100.477,164.821,57.527,160.083
C08119=1015.364,-122.035,-100.468,164.818,57.534,160.083
C08120=1015.358,-122.347,-100.459,164.814,57.542,160.084
C08121=1015.352,-122.659,-100.450,164.811,57.549,160.084
C08122=1015.347,-122.910,-100.443,164.808,57.556,160.084
C08123=1015.342,-123.159,-100.436,164.805,57.562,160.085
C08124=1015.337,-123.409,-100.429,164.803,57.567,160.085
C08125=1015.333,-123.659,-100.421,164.800,57.572,160.085
C08126=1015.327,-123.908,-100.414,164.796,57.579,160.085
C08127=1015.323,-124.158,-100.407,164.794,57.585,160.086
C08128=1015.319,-124.408,-100.400,164.791,57.591,160.086
C08129=1015.313,-124.658,-100.393,164.789,57.596,160.087
C08130=1015.309,-124.908,-100.385,164.786,57.602,160.087
C08131=1015.304,-125.158,-100.379,164.783,57.609,160.087
C08132=1015.300,-125.407,-100.372,164.780,57.614,160.087
C08133=1015.294,-125.657,-100.365,164.778,57.620,160.088
C08134=1015.290,-125.908,-100.358,164.775,57.626,160.088
C08135=1015.285,-126.157,-100.351,164.772,57.632,160.088
C08136=1015.281,-126.407,-100.344,164.769,57.638,160.089
C08137=1015.276,-126.657,-100.338,164.767,57.644,160.089
C08138=1015.271,-126.907,-100.330,164.764,57.650,160.090
C08139=1015.266,-127.157,-100.324,164.761,57.656,160.090
C08140=1015.262,-127.406,-100.316,164.758,57.661,160.090
C08141=1015.257,-127.656,-100.310,164.755,57.667,160.090
C08142=1015.253,-127.906,-100.303,164.753,57.673,160.091
C08143=1015.247,-128.155,-100.296,164.749,57.680,160.091
C08144=1015.243,-128.405,-100.289,164.747,57.684,160.091
C08145=1015.239,-128.655,-100.281,164.744,57.689,160.091
C08146=1015.236,-128.904,-100.272,164.742,57.694,160.091
C08147=1015.232,-129.154,-100.263,164.739,57.698,160.091
C08148=1015.229,-129.403,-100.253,164.736,57.701,160.091
C08149=1015.226,-129.653,-100.243,164.734,57.704,160.091
C08150=1015.224,-129.902,-100.232,164.732,57.706,160.091
C08151=1015.222,-130.152,-100.220,164.729,57.707,160.090
C08152=1015.221,-130.402,-100.209,164.726,57.708,160.090
C08153=1015.220,-130.651,-100.196,164.724,57.709,160.089
C08154=1015.219,-130.901,-100.182,164.722,57.709,160.089
C08155=1015.219,-131.151,-100.169,164.720,57.708,160.088
C08156=1015.219,-131.401,-100.154,164.718,57.707,160.087
C08157=1015.219,-131.650,-100.139,164.716,57.704,160.086
C08158=1015.220,-131.900,-100.124,164.713,57.702,160.085
C08159=1015.221,-132.150,-100.107,164.712,57.699,160.084
C08160=1015.223,-132.399,-100.090,164.710,57.696,160.083
C08161=1015.224,-132.649,-100.072,164.708,57.692,160.082
C08162=1015.227,-132.898,-100.055,164.705,57.687,160.080
C08163=1015.229,-133.148,-100.036,164.704,57.682,160.079
C08164=1015.232,-133.398,-100.017,164.703,57.676,160.078
C08165=1015.235,-133.647,-99.997,164.701,57.670,160.076
C08166=1014.993,-133.674,-100.401,164.670,58.036,160.133
C08167=1014.990,-133.424,-100.421,164.670,58.043,160.135
C08168=1014.987,-133.175,-100.440,164.673,58.048,160.136
C08169=1014.984,-132.925,-100.458,164.674,58.053,160.138
C08170=1014.982,-132.675,-100.476,164.677,58.058,160.139
C08171=1014.980,-132.426,-100.494,164.679,58.062,160.141
C08172=1014.979,-132.176,-100.511,164.680,58.066,160.142
C08173=1014.978,-131.926,-100.527,164.682,58.069,160.143
C08174=1014.977,-131.677,-100.543,164.684,58.071,160.144
C08175=1014.977,-131.427,-100.558,164.687,58.073,160.145
C08176=1014.976,-131.178,-100.573,164.688,58.074,160.145
C08177=1014.976,-130.928,-100.587,164.691,58.074,160.146
C08178=1014.977,-130.678,-100.600,164.693,58.075,160.147
C08179=1014.979,-130.429,-100.612,164.696,58.075,160.147
C08180=1014.980,-130.179,-100.624,164.698,58.074,160.148
C08181=1014.981,-129.929,-100.636,164.700,58.072,160.148
C08182=1014.984,-129.679,-100.647,164.702,58.070,160.148
C08183=1014.987,-129.430,-100.657,164.705,58.067,160.149
C08184=1014.989,-129.180,-100.667,164.707,58.064,160.149
C08185=1014.992,-128.930,-100.676,164.710,58.060,160.149
C08186=1014.996,-128.681,-100.684,164.712,58.056,160.149
C08187=1015.001,-128.432,-100.693,164.715,58.051,160.149
C08188=1015.005,-128.182,-100.700,164.718,58.046,160.148
C08189=1015.009,-127.932,-100.707,164.721,58.040,160.148
C08190=1015.014,-127.682,-100.713,164.723,58.034,160.148
C08191=1015.019,-127.433,-100.721,164.726,58.028,160.147
C08192=1015.023,-127.183,-100.727,164.729,58.023,160.147
C08193=1015.028,-126.933,-100.734,164.732,58.016,160.147
C08194=1015.033,-126.684,-100.741,164.735,58.011,160.147
C08195=1015.038,-126.433,-100.748,164.737,58.005,160.146
C08196=1015.043,-126.183,-100.755,164.739,57.999,160.146
C08197=1015.047,-125.933,-100.762,164.743,57.992,160.146
C08198=1015.052,-125.684,-100.769,164.745,57.987,160.145
C08199=1015.056,-125.434,-100.776,164.748,57.981,160.145
C08200=1015.062,-125.184,-100.782,164.751,57.975,160.145
C08201=1015.066,-124.934,-100.790,164.754,57.969,160.145
C08202=1015.071,-124.684,-100.796,164.757,57.963,160.144
C08203=1015.075,-124.434,-100.803,164.759,57.957,160.144
C08204=1015.079,-124.185,-100.811,164.762,57.951,160.143
C08205=1015.085,-123.935,-100.818,164.764,57.946,160.143
C08206=1015.089,-123.685,-100.825,164.768,57.939,160.143
C08207=1015.094,-123.435,-100.831,164.770,57.933,160.142
C08208=1015.099,-123.186,-100.839,164.773,57.928,160.142
C08209=1015.104,-122.935,-100.847,164.776,57.922,160.142
C08210=1015.108,-122.685,-100.853,164.779,57.916,160.142
C08211=1015.113,-122.436,-100.860,164.782,57.910,160.141
C08212=1015.117,-122.186,-100.867,164.784,57.904,160.141
C08213=1015.123,-121.936,-100.875,164.786,57.898,160.141
C08214=1015.127,-121.686,-100.882,164.790,57.892,160.140
C08215=1015.131,-121.436,-100.889,164.792,57.886,160.140
C08216=1015.137,-121.186,-100.896,164.795,57.880,160.140
C08217=1015.141,-120.936,-100.903,164.797,57.874,160.139
C08218=1015.146,-120.687,-100.911,164.801,57.868,160.139
C08219=1015.151,-120.438,-100.918,164.803,57.862,160.139
C08220=1015.156,-120.187,-100.925,164.806,57.856,160.138
C08221=1015.160,-119.937,-100.932,164.809,57.850,160.138
C08222=1015.165,-119.688,-100.939,164.812,57.844,160.138
C08223=1015.170,-119.437,-100.947,164.814,57.838,160.137
C08224=1015.174,-119.188,-100.954,164.818,57.832,160.137
C08225=1015.178,-118.938,-100.961,164.820,57.826,160.137
C08226=1015.184,-118.688,-100.969,164.823,57.820,160.136
C08227=1015.189,-118.406,-100.976,164.826,57.814,160.136
C08228=1015.195,-118.124,-100.985,164.829,57.807,160.136
C08229=1015.200,-117.841,-100.993,164.832,57.800,160.135
C08230=1015.206,-117.560,-101.001,164.836,57.793,160.135
C08231=1015.210,-117.310,-101.009,164.839,57.787,160.135
C08232=1015.215,-117.060,-101.017,164.842,57.781,160.134
C08233=1015.219,-116.810,-101.024,164.844,57.775,160.134
C08234=1015.224,-116.561,-101.031,164.848,57.769,160.134
C08235=1015.229,-116.310,-101.039,164.850,57.763,160.133
C08236=1015.234,-116.061,-101.046,164.852,57.756,160.133
C08237=1015.239,-115.810,-101.054,164.855,57.750,160.133
C08238=1015.244,-115.561,-101.060,164.858,57.744,160.132
C08239=1015.249,-115.311,-101.068,164.860,57.738,160.132
C08240=1015.253,-115.061,-101.076,164.864,57.732,160.132
C08241=1015.257,-114.811,-101.083,164.866,57.726,160.131
C08242=1015.263,-114.561,-101.090,164.869,57.720,160.131
C08243=1015.267,-114.312,-101.098,164.872,57.714,160.131
C08244=1015.272,-114.061,-101.105,164.875,57.708,160.130
C08245=1015.277,-113.812,-101.114,164.877,57.702,160.130
C08246=1015.282,-113.562,-101.121,164.881,57.696,160.130
C08247=1015.286,-113.312,-101.129,164.883,57.690,160.129
C08248=1015.291,-113.062,-101.136,164.887,57.684,160.129
C08249=1015.296,-112.813,-101.143,164.889,57.678,160.129
C08250=1015.301,-112.562,-101.151,164.892,57.672,160.128
C08251=1015.306,-112.313,-101.158,164.895,57.665,160.128
C08252=1015.311,-112.063,-101.167,164.897,57.659,160.127
C08253=1015.315,-111.813,-101.174,164.900,57.653,160.127
C08254=1015.320,-111.563,-101.182,164.903,57.647,160.127
C08255=1015.325,-111.313,-101.190,164.906,57.641,160.126
C08256=1015.330,-111.063,-101.197,164.909,57.635,160.126
C08257=1015.335,-110.814,-101.205,164.912,57.629,160.126
C08258=1015.340,-110.564,-101.213,164.914,57.622,160.125
C08259=1015.344,-110.314,-101.220,164.917,57.616,160.125
C08260=1015.349,-110.064,-101.228,164.920,57.610,160.125
C08261=1015.354,-109.815,-101.236,164.923,57.604,160.124
C08262=1015.359,-109.565,-101.244,164.926,57.598,160.124
C08263=1015.365,-109.232,-101.253,164.929,57.590,160.123
C08264=1015.371,-108.900,-101.264,164.934,57.581,160.123
C08265=1015.378,-108.567,-101.274,164.937,57.573,160.122
C08266=1015.385,-108.235,-101.285,164.941,57.565,160.122
C08267=1015.390,-107.985,-101.292,164.944,57.558,160.122
C08268=1015.394,-107.735,-101.300,164.947,57.553,160.121
C08269=1015.399,-107.485,-101.308,164.948,57.546,160.121
C08270=1015.404,-107.235,-101.316,164.952,57.540,160.120
C08271=1015.409,-106.985,-101.323,164.954,57.534,160.120
C08272=1015.414,-106.736,-101.332,164.958,57.528,160.120
C08273=1015.418,-106.486,-101.339,164.961,57.522,160.119
C08274=1015.424,-106.236,-101.348,164.964,57.515,160.119
C08275=1015.429,-105.986,-101.356,164.966,57.509,160.119
C08276=1015.433,-105.736,-101.363,164.968,57.503,160.118
C08277=1015.438,-105.487,-101.372,164.972,57.497,160.118
C08278=1015.442,-105.236,-101.380,164.975,57.491,160.118
C08279=1015.447,-104.987,-101.388,164.978,57.485,160.117
C08280=1015.452,-104.737,-101.396,164.980,57.478,160.117
C08281=1015.457,-104.487,-101.404,164.984,57.472,160.117
C08282=1015.462,-104.237,-101.412,164.986,57.466,160.116
C08283=1015.467,-103.988,-101.420,164.990,57.460,160.116
C08284=1015.472,-103.737,-101.428,164.991,57.453,160.115
C08285=1015.477,-103.488,-101.436,164.994,57.447,160.115
C08286=1015.482,-103.238,-101.444,164.998,57.441,160.115
C08287=1015.486,-103.014,-101.451,165.000,57.435,160.114
C08288=1015.490,-102.789,-101.459,165.003,57.430,160.114
C08289=1015.494,-102.565,-101.466,165.006,57.424,160.114
C08290=1015.499,-102.340,-101.473,165.008,57.418,160.113
C08291=1015.503,-102.116,-101.481,165.011,57.412,160.113
C08292=1015.508,-101.891,-101.488,165.013,57.408,160.113
C08293=1015.512,-101.666,-101.495,165.015,57.402,160.112
C08294=1015.517,-101.442,-101.503,165.018,57.396,160.112
C08295=1015.522,-101.192,-101.511,165.021,57.390,160.112
C08296=1015.526,-100.943,-101.519,165.023,57.383,160.111
C08297=1015.532,-100.693,-101.527,165.027,57.377,160.111
C08298=1015.537,-100.443,-101.535,165.029,57.371,160.110
C08299=1015.542,-100.193,-101.543,165.032,57.364,160.110
C08300=1015.546,-99.944,-101.552,165.035,57.358,160.109
C08301=1015.551,-99.693,-101.560,165.038,57.352,160.109
C08302=1015.556,-99.444,-101.568,165.041,57.345,160.109
C08303=1015.561,-99.194,-101.577,165.044,57.339,160.108
C08304=1015.566,-98.944,-101.584,165.047,57.333,160.108
C08305=1015.571,-98.694,-101.593,165.049,57.326,160.107
C08306=1015.576,-98.445,-101.601,165.053,57.320,160.107
C08307=1015.581,-98.194,-101.609,165.055,57.313,160.107
C08308=1015.586,-97.945,-101.617,165.058,57.307,160.106
C08309=1015.590,-97.695,-101.626,165.061,57.301,160.106
C08310=1015.595,-97.445,-101.634,165.064,57.295,160.106
C08311=1015.600,-97.195,-101.643,165.066,57.289,160.105
C08312=1015.605,-96.945,-101.651,165.070,57.282,160.105
C08313=1015.610,-96.696,-101.660,165.072,57.276,160.104
C08314=1015.615,-96.446,-101.669,165.075,57.271,160.104
C08315=1015.620,-96.196,-101.677,165.078,57.264,160.104
C08316=1015.624,-95.946,-101.686,165.080,57.258,160.103
C08317=1015.629,-95.697,-101.695,165.084,57.252,160.103
C08318=1015.634,-95.446,-101.702,165.086,57.246,160.103
C08319=1015.639,-95.196,-101.711,165.089,57.239,160.102
C08320=1015.644,-94.947,-101.720,165.092,57.233,160.102
C08321=1015.649,-94.697,-101.729,165.096,57.227,160.101
C08322=1015.654,-94.447,-101.738,165.097,57.220,160.101
C08323=1015.659,-94.198,-101.746,165.101,57.214,160.101
C08324=1015.663,-93.948,-101.755,165.104,57.208,160.100
C08325=1015.668,-93.698,-101.763,165.107,57.201,160.100
C08326=1015.674,-93.448,-101.772,165.109,57.195,160.099
C08327=1015.678,-93.198,-101.781,165.113,57.189,160.099
C08328=1015.683,-92.949,-101.789,165.115,57.182,160.098
C08329=1015.688,-92.699,-101.798,165.118,57.176,160.098
C08330=1015.693,-92.449,-101.807,165.121,57.170,160.098
C08331=1015.698,-92.199,-101.815,165.124,57.163,160.097
C08332=1015.703,-91.949,-101.824,165.126,57.158,160.097
C08333=1015.708,-91.700,-101.833,165.129,57.151,160.096
C08334=1015.713,-91.450,-101.842,165.132,57.145,160.096
C08335=1015.718,-91.200,-101.850,165.135,57.139,160.096
C08336=1015.723,-90.951,-101.859,165.138,57.132,160.095
C08337=1015.727,-90.701,-101.868,165.141,57.126,160.095
C08338=1015.733,-90.451,-101.876,165.144,57.119,160.094
C08339=1015.737,-90.201,-101.885,165.146,57.113,160.094
C08340=1015.742,-89.951,-101.894,165.150,57.106,160.094
C08341=1015.748,-89.702,-101.902,165.152,57.100,160.093
C08342=1015.752,-89.452,-101.911,165.156,57.094,160.093
C08343=1015.757,-89.202,-101.920,165.158,57.087,160.092
C08344=1015.762,-88.952,-101.929,165.161,57.081,160.092
C08345=1015.767,-88.703,-101.938,165.164,57.074,160.092
C08346=1015.773,-88.453,-101.947,165.167,57.068,160.091
C08347=1015.777,-88.203,-101.956,165.170,57.061,160.091
C08348=1015.783,-87.953,-101.964,165.172,57.056,160.090
C08349=1015.787,-87.703,-101.973,165.175,57.049,160.090
C08350=1015.792,-87.454,-101.982,165.178,57.042,160.089
C08351=1015.797,-87.203,-101.991,165.181,57.036,160.089
C08352=1015.803,-86.953,-102.000,165.184,57.029,160.088
C08353=1015.808,-86.704,-102.009,165.188,57.023,160.088
C08354=1015.813,-86.454,-102.018,165.189,57.016,160.087
C08355=1015.818,-86.174,-102.027,165.193,57.009,160.087
C08356=1015.824,-85.894,-102.037,165.197,57.002,160.087
C08357=1015.830,-85.615,-102.047,165.199,56.994,160.086
C08358=1015.836,-85.335,-102.057,165.202,56.987,160.085
C08359=1015.840,-85.085,-102.067,165.206,56.981,160.085
C08360=1015.846,-84.835,-102.075,165.209,56.974,160.085
C08361=1015.851,-84.585,-102.083,165.211,56.967,160.084
C08362=1015.856,-84.336,-102.093,165.214,56.961,160.084
C08363=1015.861,-84.086,-102.102,165.217,56.954,160.083
C08364=1015.865,-83.836,-102.111,165.219,56.948,160.083
C08365=1015.871,-83.586,-102.119,165.223,56.941,160.082
C08366=1015.876,-83.336,-102.129,165.226,56.934,160.082
C08367=1015.881,-83.086,-102.138,165.228,56.928,160.081
C08368=1015.887,-82.837,-102.146,165.232,56.922,160.081
C08369=1015.891,-82.587,-102.156,165.235,56.915,160.081
C08370=1015.897,-82.338,-102.165,165.238,56.908,160.080
C08371=1015.901,-82.088,-102.174,165.240,56.902,160.080
C08372=1015.907,-81.838,-102.182,165.243,56.895,160.079
C08373=1015.912,-81.588,-102.192,165.246,56.888,160.079
C08374=1015.917,-81.338,-102.201,165.248,56.882,160.078
C08375=1015.923,-81.088,-102.209,165.252,56.875,160.078
C08376=1015.927,-80.839,-102.219,165.255,56.868,160.077
C08377=1015.933,-80.589,-102.228,165.258,56.862,160.077
C08378=1015.938,-80.338,-102.237,165.260,56.855,160.076
C08379=1015.943,-80.089,-102.246,165.264,56.849,160.076
C08380=1015.948,-79.839,-102.255,165.266,56.842,160.075
C08381=1015.953,-79.590,-102.265,165.269,56.836,160.075
C08382=1015.957,-79.340,-102.274,165.272,56.829,160.074
C08383=1015.963,-79.090,-102.284,165.275,56.823,160.074
C08384=1015.968,-78.840,-102.293,165.278,56.816,160.074
C08385=1015.973,-78.591,-102.303,165.280,56.810,160.073
C08386=1015.978,-78.341,-102.311,165.284,56.804,160.073
C08387=1015.983,-78.091,-102.321,165.287,56.797,160.072
C08388=1015.988,-77.841,-102.330,165.289,56.791,160.072
C08389=1015.994,-77.592,-102.340,165.292,56.784,160.071
C08390=1015.998,-77.342,-102.349,165.295,56.777,160.071
C08391=1016.003,-77.092,-102.359,165.298,56.771,160.070
C08392=1016.008,-76.842,-102.369,165.301,56.764,160.070
C08393=1016.014,-76.592,-102.377,165.304,56.757,160.069
C08394=1016.018,-76.343,-102.387,165.307,56.752,160.069
C08395=1016.024,-76.093,-102.397,165.310,56.745,160.068
C08396=1016.029,-75.843,-102.406,165.313,56.738,160.068
C08397=1016.034,-75.594,-102.415,165.315,56.732,160.068
C08398=1016.039,-75.343,-102.425,165.318,56.725,160.067
C08399=1016.044,-75.094,-102.435,165.321,56.718,160.067
C08400=1016.049,-74.845,-102.444,165.324,56.712,160.066
C08401=1016.054,-74.595,-102.453,165.327,56.705,160.066
C08402=1016.059,-74.344,-102.463,165.329,56.699,160.065
C08403=1016.064,-74.095,-102.473,165.333,56.693,160.065
C08404=1016.069,-73.846,-102.483,165.335,56.686,160.064
C08405=1016.074,-73.595,-102.492,165.338,56.680,160.064
C08406=1016.079,-73.345,-102.502,165.341,56.673,160.063
C08407=1016.084,-73.096,-102.512,165.344,56.667,160.063
C08408=1016.089,-72.846,-102.522,165.347,56.660,160.062
C08409=1016.094,-72.597,-102.532,165.350,56.655,160.062
C08410=1016.100,-72.346,-102.542,165.353,56.648,160.062
C08411=1016.104,-72.097,-102.552,165.355,56.642,160.061
C08412=1016.109,-71.847,-102.561,165.358,56.635,160.061
C08413=1016.114,-71.597,-102.571,165.361,56.629,160.060
C08414=1016.119,-71.348,-102.581,165.364,56.622,160.060
C08415=1016.124,-71.098,-102.591,165.368,56.616,160.060
C08416=1016.129,-70.848,-102.601,165.370,56.610,160.059
C08417=1016.134,-70.599,-102.610,165.373,56.603,160.058
C08418=1016.140,-70.348,-102.621,165.375,56.597,160.058
C08419=1016.145,-70.071,-102.631,165.379,56.589,160.057
C08420=1016.150,-69.792,-102.643,165.382,56.582,160.057
C08421=1016.156,-69.515,-102.653,165.385,56.575,160.056
C08422=1016.162,-69.237,-102.665,165.388,56.568,160.056
C08423=1016.167,-68.987,-102.675,165.391,56.561,160.055
C08424=1016.172,-68.737,-102.685,165.393,56.555,160.055
C08425=1016.177,-68.488,-102.695,165.397,56.549,160.054
C08426=1016.182,-68.238,-102.704,165.400,56.542,160.054
C08427=1016.187,-67.988,-102.714,165.402,56.535,160.053
C08428=1016.192,-67.738,-102.724,165.406,56.529,160.053
C08429=1016.197,-67.488,-102.734,165.409,56.522,160.053
C08430=1016.202,-67.239,-102.744,165.411,56.516,160.052
C08431=1016.208,-66.989,-102.754,165.414,56.510,160.052
C08432=1016.212,-66.739,-102.764,165.416,56.503,160.051
C08433=1016.218,-66.490,-102.775,165.420,56.496,160.050
C08434=1016.223,-66.240,-102.784,165.423,56.489,160.050
C08435=1016.228,-65.990,-102.795,165.425,56.484,160.050
C08436=1016.233,-65.741,-102.804,165.428,56.477,160.049
C08437=1016.239,-65.491,-102.815,165.431,56.470,160.049
C08438=1016.244,-65.241,-102.824,165.433,56.463,160.048
C08439=1016.249,-64.991,-102.835,165.437,56.457,160.048
C08440=1016.253,-64.741,-102.845,165.440,56.450,160.047
C08441=1016.259,-64.491,-102.855,165.442,56.444,160.046
C08442=1016.263,-64.242,-102.865,165.445,56.437,160.046
C08443=1016.269,-63.992,-102.875,165.448,56.430,160.045
C08444=1016.274,-63.742,-102.885,165.451,56.424,160.045
C08445=1016.279,-63.492,-102.895,165.454,56.417,160.045
C08446=1016.285,-63.243,-102.906,165.457,56.410,160.044
C08447=1016.290,-62.993,-102.916,165.459,56.404,160.043
C08448=1016.295,-62.743,-102.926,165.462,56.397,160.043
C08449=1016.300,-62.494,-102.936,165.466,56.391,160.043
C08450=1016.305,-62.244,-102.946,165.468,56.384,160.042
C08451=1016.310,-61.994,-102.956,165.471,56.377,160.041
C08452=1016.316,-61.744,-102.966,165.474,56.371,160.041
C08453=1016.321,-61.495,-102.977,165.477,56.364,160.040
C08454=1016.326,-61.245,-102.986,165.480,56.357,160.040
C08455=1016.332,-60.995,-102.997,165.483,56.350,160.039
C08456=1016.336,-60.746,-103.006,165.486,56.343,160.039
C08457=1016.342,-60.496,-103.017,165.488,56.337,160.038
C08458=1016.348,-60.246,-103.027,165.491,56.331,160.038
C08459=1016.352,-59.997,-103.037,165.495,56.324,160.037
C08460=1016.358,-59.747,-103.047,165.498,56.317,160.037
C08461=1016.363,-59.497,-103.058,165.500,56.311,160.036
C08462=1016.367,-59.247,-103.068,165.503,56.304,160.036
C08463=1016.373,-58.997,-103.079,165.506,56.297,160.035
C08464=1016.378,-58.748,-103.089,165.509,56.290,160.035
C08465=1016.383,-58.498,-103.099,165.511,56.284,160.034
C08466=1016.389,-58.248,-103.109,165.514,56.277,160.033
C08467=1016.394,-57.999,-103.119,165.517,56.270,160.033
C08468=1016.399,-57.749,-103.130,165.521,56.263,160.032
C08469=1016.405,-57.499,-103.140,165.523,56.256,160.032
C08470=1016.411,-57.249,-103.151,165.526,56.250,160.031
C08471=1016.415,-57.000,-103.160,165.529,56.243,160.031
C08472=1016.421,-56.750,-103.171,165.532,56.236,160.030
C08473=1016.426,-56.500,-103.181,165.534,56.229,160.030
C08474=1016.431,-56.251,-103.191,165.537,56.223,160.029
C08475=1016.437,-56.001,-103.201,165.540,56.216,160.029
C08476=1016.442,-55.751,-103.212,165.543,56.209,160.028
C08477=1016.448,-55.501,-103.222,165.547,56.202,160.028
C08478=1016.452,-55.251,-103.233,165.549,56.195,160.027
C08479=1016.458,-55.002,-103.244,165.552,56.189,160.026
C08480=1016.463,-54.752,-103.254,165.554,56.181,160.026
C08481=1016.468,-54.502,-103.264,165.558,56.174,160.025
C08482=1016.474,-54.253,-103.275,165.561,56.167,160.025
C08483=1016.480,-53.976,-103.286,165.564,56.160,160.024
C08484=1016.486,-53.698,-103.297,165.566,56.153,160.023
C08485=1016.492,-53.422,-103.309,165.570,56.145,160.023
C08486=1016.498,-53.145,-103.320,165.573,56.137,160.022
C08487=1016.503,-52.896,-103.330,165.576,56.130,160.021
C08488=1016.509,-52.646,-103.341,165.579,56.124,160.021
C08489=1016.514,-52.396,-103.352,165.582,56.117,160.020
C08490=1016.519,-52.146,-103.363,165.585,56.110,160.020
C08491=1016.525,-51.896,-103.373,165.587,56.103,160.019
C08492=1016.530,-51.647,-103.383,165.590,56.096,160.018
C08493=1016.535,-51.397,-103.393,165.593,56.089,160.018
C08494=1016.541,-51.148,-103.404,165.596,56.082,160.017
C08495=1016.546,-50.898,-103.414,165.599,56.075,160.017
C08496=1016.551,-50.648,-103.426,165.601,56.069,160.016
C08497=1016.557,-50.398,-103.436,165.605,56.062,160.016
C08498=1016.562,-50.148,-103.448,165.607,56.056,160.015
C08499=1016.567,-49.899,-103.458,165.610,56.049,160.015
///RCONF 1,0,0,0,0,0,0,0,0,0,0,0,0,0,0,0,0,0,0,0,0,0,0,0
C08500=1016.572,-49.649,-103.469,165.613,56.042,160.014
C08501=1016.577,-49.399,-103.480,165.616,56.036,160.014
C08502=1016.582,-49.149,-103.491,165.619,56.029,160.013
C08503=1016.588,-48.900,-103.502,165.622,56.022,160.013
C08504=1016.593,-48.649,-103.513,165.624,56.016,160.012
C08505=1016.599,-48.400,-103.524,165.627,56.009,160.011
C08506=1016.603,-48.151,-103.535,165.630,56.002,160.011
C08507=1016.609,-47.901,-103.546,165.632,55.996,160.010
C08508=1016.613,-47.651,-103.556,165.636,55.989,160.010
C08509=1016.619,-47.401,-103.567,165.639,55.982,160.009
C08510=1016.624,-47.152,-103.579,165.641,55.976,160.009
C08511=1016.630,-46.902,-103.590,165.644,55.969,160.008
C08512=1016.635,-46.652,-103.600,165.647,55.962,160.008
C08513=1016.640,-46.402,-103.611,165.649,55.956,160.007
C08514=1016.645,-46.152,-103.623,165.652,55.949,160.006
C08515=1016.651,-45.904,-103.633,165.656,55.942,160.006
C08516=1016.656,-45.654,-103.645,165.659,55.935,160.005
C08517=1016.661,-45.404,-103.655,165.661,55.929,160.005
C08518=1016.666,-45.154,-103.666,165.664,55.922,160.004
C08519=1016.672,-44.904,-103.677,165.667,55.915,160.004
C08520=1016.677,-44.655,-103.689,165.669,55.909,160.003
C08521=1016.682,-44.405,-103.700,165.673,55.902,160.002
C08522=1016.687,-44.155,-103.711,165.676,55.895,160.002
C08523=1016.693,-43.906,-103.722,165.679,55.888,160.001
C08524=1016.698,-43.655,-103.733,165.681,55.882,160.001
C08525=1016.704,-43.406,-103.744,165.684,55.874,160.000
C08526=1016.709,-43.156,-103.755,165.687,55.867,159.999
C08527=1016.714,-42.907,-103.766,165.689,55.861,159.999
C08528=1016.719,-42.657,-103.777,165.692,55.854,159.998
C08529=1016.725,-42.407,-103.788,165.695,55.847,159.998
C08530=1016.730,-42.158,-103.800,165.698,55.841,159.997
C08531=1016.736,-41.908,-103.811,165.701,55.834,159.997
C08532=1016.741,-41.658,-103.822,165.704,55.827,159.996
C08533=1016.747,-41.409,-103.833,165.707,55.821,159.996
C08534=1016.752,-41.159,-103.844,165.710,55.813,159.995
C08535=1016.757,-40.909,-103.855,165.712,55.807,159.994
C08536=1016.762,-40.659,-103.866,165.715,55.800,159.994
C08537=1016.768,-40.410,-103.877,165.718,55.793,159.993
C08538=1016.773,-40.160,-103.888,165.721,55.786,159.993
C08539=1016.778,-39.910,-103.899,165.723,55.779,159.992
C08540=1016.783,-39.660,-103.911,165.726,55.772,159.991
C08541=1016.789,-39.411,-103.922,165.729,55.765,159.991
C08542=1016.794,-39.161,-103.933,165.731,55.759,159.990
C08543=1016.800,-38.912,-103.945,165.735,55.752,159.989
C08544=1016.805,-38.662,-103.956,165.738,55.745,159.989
C08545=1016.810,-38.413,-103.968,165.740,55.739,159.988
C08546=1016.815,-38.163,-103.979,165.743,55.732,159.988
C08547=1016.821,-37.886,-103.992,165.746,55.725,159.987
C08548=1016.827,-37.610,-104.005,165.750,55.717,159.987
C08549=1016.833,-37.333,-104.017,165.753,55.710,159.986
C08550=1016.839,-37.057,-104.030,165.755,55.702,159.985
C08551=1016.844,-36.807,-104.042,165.758,55.696,159.985
C08552=1016.849,-36.557,-104.053,165.761,55.689,159.984
C08553=1016.855,-36.307,-104.065,165.764,55.682,159.983
C08554=1016.860,-36.057,-104.076,165.767,55.676,159.983
C08555=1016.866,-35.808,-104.088,165.769,55.669,159.982
C08556=1016.871,-35.559,-104.100,165.772,55.662,159.982
C08557=1016.876,-35.309,-104.111,165.776,55.656,159.981
C08558=1016.881,-35.059,-104.122,165.778,55.649,159.980
C08559=1016.887,-34.810,-104.134,165.780,55.642,159.980
C08560=1016.892,-34.560,-104.146,165.784,55.635,159.979
C08561=1016.897,-34.310,-104.157,165.786,55.628,159.979
C08562=1016.902,-34.060,-104.169,165.789,55.622,159.978
C08563=1016.908,-33.811,-104.180,165.792,55.615,159.977
C08564=1016.913,-33.561,-104.192,165.795,55.608,159.977
C08565=1016.918,-33.311,-104.203,165.797,55.602,159.976
C08566=1016.923,-33.062,-104.215,165.800,55.594,159.976
C08567=1016.929,-32.812,-104.227,165.803,55.587,159.975
C08568=1016.935,-32.562,-104.238,165.806,55.581,159.974
C08569=1016.940,-32.312,-104.250,165.809,55.574,159.974
C08570=1016.945,-32.063,-104.262,165.812,55.567,159.973
C08571=1016.950,-31.814,-104.273,165.814,55.560,159.972
C08572=1016.957,-31.563,-104.285,165.817,55.554,159.972
C08573=1016.962,-31.314,-104.297,165.820,55.547,159.971
C08574=1016.967,-31.064,-104.308,165.823,55.540,159.971
C08575=1016.972,-30.815,-104.320,165.825,55.534,159.970
C08576=1016.977,-30.565,-104.332,165.828,55.526,159.969
C08577=1016.984,-30.315,-104.343,165.831,55.519,159.969
C08578=1016.989,-30.065,-104.355,165.833,55.513,159.968
C08579=1016.994,-29.816,-104.367,165.836,55.505,159.967
C08580=1016.999,-29.566,-104.378,165.839,55.499,159.967
C08581=1017.005,-29.316,-104.391,165.843,55.492,159.966
C08582=1017.011,-29.067,-104.402,165.845,55.485,159.966
C08583=1017.016,-28.817,-104.413,165.847,55.478,159.965
C08584=1017.021,-28.568,-104.426,165.851,55.471,159.964
C08585=1017.026,-28.318,-104.437,165.854,55.464,159.964
C08586=1017.032,-28.068,-104.450,165.856,55.457,159.963
C08587=1017.038,-27.819,-104.460,165.859,55.451,159.962
C08588=1017.043,-27.570,-104.473,165.862,55.444,159.962
C08589=1017.048,-27.319,-104.485,165.864,55.437,159.961
C08590=1017.053,-27.070,-104.497,165.867,55.431,159.961
C08591=1017.058,-26.820,-104.509,165.871,55.424,159.960
C08592=1017.064,-26.570,-104.521,165.872,55.417,159.959
C08593=1017.069,-26.321,-104.533,165.876,55.410,159.959
C08594=1017.074,-26.071,-104.545,165.879,55.403,159.958
C08595=1017.080,-25.821,-104.557,165.881,55.397,159.958
C08596=1017.085,-25.571,-104.569,165.884,55.390,159.957
C08597=1017.090,-25.322,-104.581,165.886,55.384,159.956
C08598=1017.096,-25.072,-104.594,165.889,55.376,159.956
C08599=1017.101,-24.822,-104.605,165.892,55.370,159.955
C08600=1017.107,-24.573,-104.617,165.894,55.363,159.954
C08601=1017.113,-24.323,-104.630,165.898,55.356,159.954
C08602=1017.117,-24.073,-104.642,165.901,55.350,159.953
C08603=1017.122,-23.824,-104.654,165.903,55.343,159.953
C08604=1017.128,-23.574,-104.667,165.906,55.336,159.952
C08605=1017.133,-23.324,-104.678,165.909,55.329,159.951
C08606=1017.138,-23.075,-104.690,165.911,55.323,159.951
C08607=1017.144,-22.825,-104.703,165.915,55.316,159.950
C08608=1017.150,-22.576,-104.715,165.917,55.308,159.949
C08609=1017.155,-22.326,-104.727,165.919,55.302,159.949
C08610=1017.160,-22.076,-104.739,165.923,55.295,159.948
C08611=1017.166,-21.799,-104.753,165.925,55.288,159.947
C08612=1017.172,-21.522,-104.767,165.929,55.280,159.947
C08613=1017.178,-21.244,-104.780,165.932,55.273,159.946
C08614=1017.184,-20.967,-104.793,165.935,55.265,159.945
C08615=1017.190,-20.716,-104.805,165.938,55.258,159.945
C08616=1017.195,-20.467,-104.818,165.940,55.251,159.944
C08617=1017.200,-20.218,-104.830,165.943,55.244,159.943
C08618=1017.206,-19.968,-104.843,165.946,55.238,159.943
C08619=1017.211,-19.718,-104.854,165.949,55.230,159.942
C08620=1017.217,-19.468,-104.867,165.951,55.224,159.941
C08621=1017.222,-19.219,-104.879,165.954,55.217,159.941
C08622=1017.228,-18.969,-104.892,165.957,55.210,159.940
C08623=1017.233,-18.720,-104.904,165.959,55.203,159.939
C08624=1017.239,-18.471,-104.916,165.962,55.197,159.939
C08625=1017.244,-18.220,-104.928,165.965,55.189,159.938
C08626=1017.249,-17.971,-104.940,165.967,55.183,159.937
C08627=1017.255,-17.721,-104.953,165.970,55.175,159.937
C08628=1017.260,-17.472,-104.965,165.973,55.169,159.936
C08629=1017.266,-17.222,-104.978,165.977,55.162,159.936
C08630=1017.271,-16.973,-104.990,165.978,55.155,159.935
C08631=1017.277,-16.722,-105.002,165.982,55.148,159.934
C08632=1017.282,-16.473,-105.014,165.984,55.141,159.933
C08633=1017.288,-16.223,-105.027,165.987,55.134,159.933
C08634=1017.293,-15.974,-105.039,165.990,55.128,159.932
C08635=1017.298,-15.724,-105.052,165.993,55.120,159.931
C08636=1017.304,-15.474,-105.064,165.995,55.114,159.931
C08637=1017.310,-15.225,-105.077,165.998,55.107,159.930
C08638=1017.314,-14.975,-105.090,166.000,55.101,159.930
C08639=1017.320,-14.725,-105.102,166.004,55.094,159.929
C08640=1017.325,-14.476,-105.115,166.006,55.087,159.928
C08641=1017.331,-14.226,-105.127,166.009,55.080,159.928
C08642=1017.336,-13.977,-105.140,166.012,55.074,159.927
C08643=1017.341,-13.727,-105.153,166.014,55.066,159.926
C08644=1017.347,-13.478,-105.166,166.017,55.060,159.926
C08645=1017.353,-13.228,-105.178,166.020,55.053,159.925
C08646=1017.357,-12.979,-105.191,166.022,55.047,159.924
C08647=1017.363,-12.729,-105.204,166.025,55.039,159.924
C08648=1017.368,-12.479,-105.216,166.028,55.033,159.923
C08649=1017.374,-12.229,-105.229,166.031,55.026,159.922
C08650=1017.379,-11.979,-105.241,166.033,55.019,159.922
C08651=1017.384,-11.730,-105.254,166.036,55.012,159.921
C08652=1017.390,-11.481,-105.267,166.039,55.006,159.921
C08653=1017.395,-11.231,-105.280,166.042,54.998,159.920
C08654=1017.401,-10.981,-105.293,166.044,54.992,159.919
C08655=1017.406,-10.732,-105.305,166.047,54.985,159.919
C08656=1017.411,-10.482,-105.318,166.050,54.978,159.918
C08657=1017.417,-10.232,-105.331,166.052,54.972,159.917
C08658=1017.422,-9.983,-105.343,166.055,54.964,159.916
C08659=1017.428,-9.733,-105.357,166.058,54.957,159.916
C08660=1017.433,-9.484,-105.369,166.061,54.951,159.915
C08661=1017.438,-9.234,-105.382,166.063,54.944,159.914
C08662=1017.444,-8.984,-105.395,166.067,54.937,159.914
C08663=1017.450,-8.735,-105.407,166.068,54.930,159.913
C08664=1017.455,-8.485,-105.421,166.072,54.923,159.912
C08665=1017.461,-8.235,-105.433,166.074,54.917,159.912
C08666=1017.465,-7.986,-105.446,166.077,54.909,159.911
C08667=1017.471,-7.736,-105.459,166.080,54.903,159.910
C08668=1017.477,-7.487,-105.471,166.082,54.896,159.909
C08669=1017.482,-7.237,-105.485,166.085,54.889,159.909
C08670=1017.488,-6.987,-105.497,166.088,54.882,159.908
C08671=1017.493,-6.738,-105.510,166.090,54.875,159.907
C08672=1017.499,-6.489,-105.523,166.093,54.868,159.907
C08673=1017.505,-6.239,-105.536,166.096,54.861,159.906
C08674=1017.509,-5.989,-105.549,166.098,54.854,159.905
C08675=1017.516,-5.710,-105.563,166.102,54.846,159.905
C08676=1017.522,-5.430,-105.577,166.105,54.839,159.904
C08677=1017.529,-5.151,-105.592,166.108,54.831,159.903
C08678=1017.534,-4.871,-105.607,166.111,54.823,159.902
C08679=1017.540,-4.622,-105.619,166.114,54.816,159.902
C08680=1017.546,-4.372,-105.632,166.116,54.809,159.901
C08681=1017.551,-4.123,-105.645,166.119,54.803,159.900
C08682=1017.556,-3.873,-105.659,166.121,54.796,159.900
C08683=1017.561,-3.624,-105.672,166.125,54.790,159.899
C08684=1017.566,-3.373,-105.685,166.126,54.783,159.898
C08685=1017.573,-3.124,-105.698,166.130,54.776,159.898
C08686=1017.578,-2.874,-105.712,166.132,54.770,159.897
C08687=1017.583,-2.625,-105.725,166.135,54.762,159.896
C08688=1017.588,-2.375,-105.738,166.138,54.756,159.896
C08689=1017.594,-2.126,-105.752,166.140,54.749,159.895
C08690=1017.599,-1.877,-105.765,166.143,54.742,159.894
C08691=1017.604,-1.627,-105.778,166.145,54.736,159.894
C08692=1017.610,-1.377,-105.792,166.149,54.729,159.893
C08693=1017.615,-1.127,-105.805,166.150,54.722,159.892
C08694=1017.620,-0.878,-105.818,166.154,54.715,159.892
C08695=1017.626,-0.628,-105.831,166.156,54.709,159.891
C08696=1017.631,-0.379,-105.845,166.159,54.701,159.890
C08697=1017.637,-0.129,-105.858,166.161,54.695,159.889
C08698=1017.642,0.120,-105.871,166.164,54.689,159.889
C08699=1017.647,0.370,-105.885,166.167,54.681,159.888
C08700=1017.652,0.620,-105.898,166.170,54.675,159.887
C08701=1017.658,0.870,-105.912,166.173,54.668,159.887
C08702=1017.664,1.119,-105.925,166.175,54.661,159.886
C08703=1017.669,1.368,-105.938,166.178,54.655,159.886
C08704=1017.674,1.618,-105.952,166.180,54.648,159.885
C08705=1017.680,1.867,-105.966,166.183,54.641,159.884
C08706=1017.686,2.117,-105.978,166.186,54.634,159.884
C08707=1017.691,2.367,-105.992,166.188,54.627,159.883
C08708=1017.696,2.616,-106.006,166.192,54.621,159.882
C08709=1017.701,2.866,-106.019,166.193,54.614,159.881
C08710=1017.707,3.116,-106.033,166.197,54.607,159.881
C08711=1017.713,3.365,-106.046,166.198,54.600,159.880
C08712=1017.718,3.615,-106.059,166.202,54.593,159.879
C08713=1017.723,3.864,-106.073,166.205,54.586,159.878
C08714=1017.728,4.113,-106.087,166.207,54.580,159.878
C08715=1017.734,4.363,-106.099,166.210,54.572,159.877
C08716=1017.740,4.613,-106.113,166.212,54.566,159.876
C08717=1017.745,4.863,-106.127,166.215,54.559,159.876
C08718=1017.751,5.112,-106.141,166.218,54.552,159.875
C08719=1017.756,5.362,-106.154,166.220,54.545,159.874
C08720=1017.761,5.611,-106.167,166.223,54.538,159.874
C08721=1017.767,5.860,-106.181,166.225,54.531,159.873
C08722=1017.772,6.110,-106.194,166.229,54.525,159.872
C08723=1017.778,6.360,-106.208,166.231,54.517,159.871
C08724=1017.783,6.610,-106.221,166.234,54.511,159.871
C08725=1017.789,6.859,-106.235,166.237,54.504,159.870
C08726=1017.795,7.109,-106.249,166.239,54.497,159.869
C08727=1017.800,7.359,-106.262,166.242,54.490,159.868
C08728=1017.805,7.608,-106.276,166.245,54.483,159.868
C08729=1017.812,7.858,-106.289,166.247,54.476,159.867
C08730=1017.816,8.107,-106.302,166.250,54.469,159.866
C08731=1017.822,8.356,-106.316,166.252,54.463,159.866
C08732=1017.827,8.606,-106.329,166.255,54.455,159.865
C08733=1017.833,8.856,-106.343,166.258,54.449,159.864
C08734=1017.839,9.105,-106.357,166.260,54.442,159.863
C08735=1017.844,9.355,-106.370,166.263,54.434,159.863
C08736=1017.850,9.604,-106.384,166.266,54.428,159.862
C08737=1017.855,9.854,-106.398,166.268,54.421,159.861
C08738=1017.861,10.103,-106.412,166.271,54.414,159.861
C08739=1017.867,10.385,-106.427,166.274,54.406,159.860
C08740=1017.873,10.666,-106.442,166.278,54.398,159.859
C08741=1017.879,10.948,-106.458,166.280,54.390,159.858
C08742=1017.885,11.229,-106.473,166.283,54.383,159.857
C08743=1017.891,11.478,-106.487,166.286,54.376,159.856
C08744=1017.896,11.728,-106.500,166.289,54.368,159.856
C08745=1017.903,11.977,-106.514,166.291,54.362,159.855
C08746=1017.908,12.227,-106.528,166.294,54.355,159.854
C08747=1017.914,12.476,-106.541,166.297,54.347,159.853
C08748=1017.919,12.726,-106.555,166.299,54.341,159.853
C08749=1017.925,12.975,-106.569,166.302,54.334,159.852
C08750=1017.930,13.225,-106.582,166.305,54.326,159.851
C08751=1017.936,13.474,-106.596,166.307,54.320,159.851
C08752=1017.941,13.724,-106.611,166.310,54.313,159.850
C08753=1017.946,13.974,-106.625,166.312,54.306,159.849
C08754=1017.952,14.223,-106.638,166.315,54.299,159.848
C08755=1017.957,14.473,-106.652,166.318,54.293,159.848
C08756=1017.963,14.722,-106.666,166.320,54.286,159.847
C08757=1017.968,14.972,-106.680,166.323,54.279,159.846
C08758=1017.974,15.222,-106.694,166.326,54.272,159.845
C08759=1017.979,15.471,-106.708,166.327,54.265,159.844
C08760=1017.985,15.721,-106.722,166.331,54.258,159.844
C08761=1017.991,15.970,-106.736,166.334,54.251,159.843
C08762=1017.997,16.220,-106.750,166.336,54.245,159.843
C08763=1018.002,16.469,-106.764,166.339,54.237,159.842
C08764=1018.007,16.719,-106.779,166.341,54.231,159.841
C08765=1018.012,16.969,-106.793,166.344,54.224,159.840
C08766=1018.018,17.219,-106.807,166.346,54.217,159.839
C08767=1018.024,17.467,-106.821,166.349,54.210,159.839
C08768=1018.029,17.717,-106.835,166.351,54.203,159.838
C08769=1018.035,17.967,-106.849,166.355,54.197,159.837
C08770=1018.040,18.216,-106.863,166.358,54.189,159.837
C08771=1018.046,18.466,-106.877,166.359,54.183,159.836
C08772=1018.051,18.715,-106.890,166.363,54.176,159.835
C08773=1018.057,18.964,-106.905,166.365,54.169,159.834
C08774=1018.062,19.214,-106.919,166.368,54.162,159.834
C08775=1018.067,19.464,-106.933,166.370,54.155,159.833
C08776=1018.073,19.713,-106.948,166.373,54.148,159.832
C08777=1018.079,19.963,-106.962,166.375,54.142,159.831
C08778=1018.084,20.213,-106.977,166.378,54.135,159.831
C08779=1018.089,20.462,-106.990,166.380,54.128,159.830
C08780=1018.095,20.711,-107.005,166.383,54.121,159.829
C08781=1018.100,20.961,-107.019,166.387,54.114,159.829
C08782=1018.105,21.211,-107.033,166.389,54.108,159.828
C08783=1018.111,21.460,-107.048,166.392,54.100,159.827
C08784=1018.116,21.709,-107.062,166.394,54.094,159.826
C08785=1018.122,21.960,-107.076,166.397,54.087,159.825
C08786=1018.127,22.209,-107.091,166.399,54.080,159.825
C08787=1018.133,22.459,-107.105,166.402,54.073,159.824
C08788=1018.139,22.707,-107.120,166.404,54.066,159.823
C08789=1018.144,22.957,-107.134,166.407,54.060,159.823
C08790=1018.149,23.207,-107.148,166.409,54.053,159.822
C08791=1018.155,23.456,-107.163,166.413,54.046,159.821
C08792=1018.161,23.706,-107.177,166.414,54.039,159.820
C08793=1018.166,23.956,-107.191,166.417,54.032,159.819
C08794=1018.171,24.205,-107.206,166.421,54.025,159.819
C08795=1018.177,24.455,-107.220,166.423,54.018,159.818
C08796=1018.183,24.704,-107.234,166.426,54.011,159.817
C08797=1018.189,24.954,-107.248,166.428,54.005,159.817
C08798=1018.194,25.203,-107.264,166.431,53.998,159.816
C08799=1018.199,25.453,-107.278,166.433,53.991,159.815
C08800=1018.205,25.702,-107.291,166.436,53.984,159.814
C08801=1018.210,25.951,-107.306,166.438,53.977,159.813
C08802=1018.216,26.202,-107.321,166.441,53.970,159.813
C08803=1018.223,26.484,-107.337,166.444,53.963,159.812
C08804=1018.228,26.767,-107.354,166.447,53.954,159.811
C08805=1018.235,27.050,-107.370,166.450,53.947,159.810
C08806=1018.240,27.333,-107.387,166.453,53.939,159.809
C08807=1018.246,27.582,-107.401,166.456,53.932,159.809
C08808=1018.251,27.832,-107.416,166.458,53.925,159.808
C08809=1018.257,28.081,-107.431,166.461,53.918,159.807
C08810=1018.262,28.331,-107.445,166.464,53.912,159.806
C08811=1018.268,28.580,-107.460,166.466,53.905,159.806
C08812=1018.273,28.829,-107.475,166.468,53.898,159.805
C08813=1018.279,29.080,-107.489,166.472,53.891,159.804
C08814=1018.284,29.329,-107.504,166.474,53.884,159.803
C08815=1018.290,29.578,-107.519,166.477,53.878,159.803
C08816=1018.295,29.828,-107.533,166.479,53.871,159.802
C08817=1018.301,30.078,-107.548,166.482,53.863,159.801
C08818=1018.306,30.327,-107.563,166.484,53.857,159.800
C08819=1018.311,30.576,-107.577,166.487,53.850,159.800
C08820=1018.317,30.826,-107.592,166.489,53.843,159.799
C08821=1018.323,31.075,-107.607,166.493,53.837,159.798
C08822=1018.328,31.325,-107.622,166.495,53.830,159.797
C08823=1018.333,31.574,-107.636,166.498,53.822,159.796
C08824=1018.338,31.823,-107.652,166.500,53.816,159.796
C08825=1018.345,32.074,-107.666,166.503,53.809,159.795
C08826=1018.350,32.323,-107.681,166.505,53.802,159.794
C08827=1018.355,32.572,-107.696,166.508,53.795,159.794
C08828=1018.361,32.822,-107.711,166.510,53.789,159.793
C08829=1018.366,33.071,-107.725,166.513,53.781,159.792
C08830=1018.372,33.321,-107.740,166.516,53.775,159.791
C08831=1018.378,33.570,-107.755,166.518,53.768,159.790
C08832=1018.383,33.820,-107.770,166.520,53.761,159.790
C08833=1018.388,34.069,-107.784,166.523,53.754,159.789
C08834=1018.394,34.319,-107.800,166.526,53.748,159.788
C08835=1018.400,34.568,-107.814,166.529,53.740,159.787
C08836=1018.405,34.817,-107.829,166.531,53.733,159.786
C08837=1018.411,35.068,-107.844,166.534,53.727,159.786
C08838=1018.416,35.317,-107.859,166.536,53.720,159.785
C08839=1018.422,35.566,-107.873,166.539,53.713,159.784
C08840=1018.427,35.816,-107.889,166.542,53.705,159.783
C08841=1018.433,36.065,-107.903,166.544,53.699,159.783
C08842=1018.438,36.315,-107.918,166.547,53.692,159.782
C08843=1018.444,36.564,-107.933,166.549,53.685,159.781
C08844=1018.449,36.814,-107.948,166.552,53.678,159.780
C08845=1018.455,37.064,-107.964,166.555,53.672,159.780
C08846=1018.460,37.313,-107.979,166.558,53.664,159.779
C08847=1018.465,37.554,-107.994,166.560,53.658,159.778
C08848=1018.470,37.795,-108.008,166.562,53.651,159.777
C08849=1018.475,38.036,-108.022,166.564,53.645,159.777
C08850=1018.481,38.277,-108.037,166.567,53.638,159.776
C08851=1018.487,38.518,-108.051,166.570,53.632,159.775
C08852=1018.492,38.759,-108.066,166.572,53.626,159.774
C08853=1018.498,39.000,-108.081,166.574,53.619,159.774
C08854=1018.502,39.242,-108.095,166.578,53.612,159.773
C08855=1018.508,39.491,-108.110,166.580,53.605,159.772
C08856=1018.513,39.740,-108.126,166.583,53.598,159.771
C08857=1018.519,39.990,-108.141,166.585,53.592,159.771
C08858=1018.524,40.239,-108.156,166.588,53.585,159.770
C08859=1018.530,40.489,-108.171,166.590,53.578,159.769
C08860=1018.535,40.738,-108.187,166.593,53.571,159.768
C08861=1018.540,40.988,-108.202,166.595,53.564,159.768
C08862=1018.546,41.237,-108.217,166.598,53.557,159.767
C08863=1018.551,41.486,-108.233,166.600,53.550,159.766
C08864=1018.557,41.736,-108.248,166.604,53.544,159.765
C08865=1018.562,41.985,-108.263,166.606,53.537,159.764
C08866=1018.569,42.235,-108.278,166.609,53.530,159.764
C08867=1018.575,42.535,-108.297,166.611,53.522,159.763
C08868=1018.581,42.835,-108.315,166.615,53.513,159.762
C08869=1018.587,43.135,-108.334,166.618,53.506,159.761
C08870=1018.594,43.434,-108.353,166.622,53.498,159.760
C08871=1018.599,43.683,-108.368,166.623,53.491,159.759
C08872=1018.604,43.932,-108.383,166.625,53.484,159.758
C08873=1018.610,44.182,-108.399,166.629,53.478,159.758
C08874=1018.615,44.431,-108.415,166.631,53.471,159.757
C08875=1018.621,44.681,-108.430,166.634,53.464,159.756
C08876=1018.626,44.930,-108.445,166.636,53.457,159.756
C08877=1018.632,45.180,-108.461,166.639,53.451,159.755
C08878=1018.636,45.429,-108.477,166.642,53.444,159.754
C08879=1018.642,45.679,-108.493,166.644,53.437,159.753
C08880=1018.647,45.928,-108.508,166.647,53.431,159.753
C08881=1018.653,46.178,-108.524,166.649,53.424,159.752
C08882=1018.658,46.427,-108.539,166.651,53.417,159.751
C08883=1018.663,46.677,-108.555,166.655,53.411,159.750
C08884=1018.669,46.926,-108.570,166.657,53.404,159.749
C08885=1018.674,47.176,-108.586,166.660,53.397,159.749
C08886=1018.680,47.425,-108.602,166.662,53.390,159.748
C08887=1018.685,47.675,-108.617,166.665,53.383,159.747
C08888=1018.691,47.923,-108.633,166.667,53.376,159.746
C08889=1018.696,48.173,-108.649,166.670,53.370,159.746
C08890=1018.701,48.423,-108.664,166.673,53.363,159.745
C08891=1018.707,48.672,-108.680,166.675,53.356,159.744
C08892=1018.712,48.921,-108.695,166.678,53.350,159.743
C08893=1018.717,49.172,-108.711,166.680,53.343,159.742
C08894=1018.722,49.420,-108.727,166.683,53.336,159.742
C08895=1018.728,49.670,-108.743,166.686,53.329,159.741
C08896=1018.733,49.919,-108.758,166.688,53.323,159.740
C08897=1018.739,50.169,-108.774,166.691,53.315,159.739
C08898=1018.745,50.419,-108.790,166.693,53.309,159.738
C08899=1018.750,50.667,-108.806,166.696,53.302,159.738
C08900=1018.756,50.917,-108.821,166.698,53.295,159.737
C08901=1018.761,51.167,-108.836,166.701,53.288,159.736
C08902=1018.767,51.416,-108.853,166.703,53.281,159.735
C08903=1018.772,51.665,-108.868,166.707,53.275,159.735
C08904=1018.778,51.915,-108.884,166.709,53.268,159.734
C08905=1018.783,52.165,-108.900,166.712,53.261,159.733
C08906=1018.788,52.414,-108.915,166.714,53.254,159.732
C08907=1018.794,52.663,-108.932,166.717,53.247,159.732
C08908=1018.799,52.913,-108.947,166.719,53.241,159.731
C08909=1018.805,53.162,-108.963,166.722,53.233,159.730
C08910=1018.810,53.412,-108.979,166.724,53.227,159.729
C08911=1018.816,53.661,-108.994,166.726,53.220,159.728
C08912=1018.821,53.911,-109.010,166.730,53.213,159.728
C08913=1018.827,54.159,-109.026,166.732,53.206,159.727
C08914=1018.832,54.409,-109.041,166.735,53.199,159.726
C08915=1018.838,54.659,-109.058,166.737,53.192,159.725
C08916=1018.843,54.908,-109.073,166.740,53.185,159.724
C08917=1018.849,55.157,-109.089,166.742,53.178,159.723
C08918=1018.855,55.407,-109.105,166.745,53.172,159.723
C08919=1018.860,55.656,-109.121,166.747,53.165,159.722
C08920=1018.865,55.906,-109.137,166.751,53.158,159.721
C08921=1018.871,56.155,-109.153,166.753,53.151,159.720
C08922=1018.876,56.405,-109.168,166.756,53.144,159.720
C08923=1018.882,56.654,-109.184,166.758,53.137,159.719
C08924=1018.888,56.904,-109.200,166.761,53.130,159.718
C08925=1018.893,57.153,-109.216,166.763,53.124,159.717
C08926=1018.899,57.403,-109.231,166.766,53.117,159.716
C08927=1018.905,57.652,-109.248,166.769,53.110,159.716
C08928=1018.910,57.901,-109.263,166.771,53.103,159.715
C08929=1018.916,58.151,-109.279,166.774,53.096,159.714
C08930=1018.921,58.401,-109.295,166.776,53.089,159.713
C08931=1018.927,58.683,-109.313,166.779,53.081,159.712
C08932=1018.934,58.966,-109.331,166.783,53.073,159.711
C08933=1018.940,59.248,-109.349,166.786,53.065,159.710
C08934=1018.946,59.531,-109.367,166.788,53.058,159.709
C08935=1018.952,59.781,-109.383,166.792,53.050,159.709
C08936=1018.957,60.031,-109.399,166.794,53.044,159.708
C08937=1018.963,60.279,-109.415,166.797,53.036,159.707
C08938=1018.969,60.529,-109.431,166.799,53.030,159.706
